LIN {X 0,Y 362.1,Z 510.041,A -85,B 0,C 180,E1 -13379.691,E2 -13379.691} C_VEL
LIN {X 0,Y 361.308,Z 518.217,A -85,B 0,C 180,E1 -13381.227,E2 -13381.227} C_VEL
LIN {X 0,Y 359.207,Z 536.983,A -85,B 0,C 180,E1 -13384.658,E2 -13384.658} C_VEL
LIN {X 0,Y 359.602,Z 541.842,A -85,B 0,C 180,E1 -13385.074,E2 -13385.074} C_VEL
LIN {X 0,Y 360.933,Z 553.52,A -85,B 0,C 180,E1 -13385.902,E2 -13385.902} C_VEL
LIN {X 0,Y 363.229,Z 569.599,A -85,B 0,C 180,E1 -13386.676,E2 -13386.676} C_VEL
LIN {X 0,Y 364.954,Z 589.975,A -85,B 0,C 180,E1 -13387.487,E2 -13387.487} C_VEL
LIN {X 0,Y 365.399,Z 602.018,A -85,B 0,C 180,E1 -13387.902,E2 -13387.902} C_VEL
LIN {X 0,Y 363.82,Z 641.826,A -85,B 0,C 180,E1 -13388.948,E2 -13388.948} C_VEL
LIN {X 0,Y 363.382,Z 660.329,A -85,B 0,C 180,E1 -13389.366,E2 -13389.366} C_VEL
LIN {X 0,Y 362.094,Z 683.326,A -85,B 0,C 180,E1 -13390.216,E2 -13390.216} C_VEL
LIN {X 0,Y 360.889,Z 696.981,A -85,B 0,C 180,E1 -13390.96,E2 -13390.96} C_VEL
LIN {X 0,Y 359.746,Z 709.851,A -85,B 0,C 180,E1 -13391.931,E2 -13391.931} C_VEL
LIN {X 0,Y 358.479,Z 721.302,A -85,B 0,C 180,E1 -13393.043,E2 -13393.043} C_VEL
LIN {X 0,Y 357.211,Z 731.941,A -85,B 0,C 180,E1 -13394.329,E2 -13394.329} C_VEL
LIN {X 0,Y 356.095,Z 741.238,A -85,B 0,C 180,E1 -13395.716,E2 -13395.716} C_VEL
LIN {X 0,Y 355.187,Z 750.5,A -85,B 0,C 180,E1 -13397.427,E2 -13397.427} C_VEL
LIN {X 0,Y 354.364,Z 757.955,A -85,B 0,C 180,E1 -13399.138,E2 -13399.138} C_VEL
LIN {X 0,Y 353.848,Z 763.907,A -85,B 0,C 180,E1 -13400.855,E2 -13400.855} C_VEL
LIN {X 0,Y 353.526,Z 768.592,A -85,B 0,C 180,E1 -13402.574,E2 -13402.574} C_VEL
LIN {X 0,Y 353.412,Z 772.146,A -85,B 0,C 180,E1 -13404.292,E2 -13404.292} C_VEL
LIN {X 0,Y 353.428,Z 773.933,A -85,B 0,C 180,E1 -13405.436,E2 -13405.436} C_VEL
LIN {X 0,Y 353.398,Z 775.272,A -85,B 0,C 180,E1 -13406.578,E2 -13406.578} C_VEL
LIN {X 0,Y 353.5,Z 776.131,A -85,B 0,C 180,E1 -13407.719,E2 -13407.719} C_VEL
LIN {X 0,Y 353.555,Z 776.567,A -85,B 0,C 180,E1 -13408.859,E2 -13408.859} C_VEL
LIN {X 0,Y 353.604,Z 776.578,A -85,B 0,C 180,E1 -13409.998,E2 -13409.998} C_VEL
LIN {X 0,Y 353.57,Z 776.1,A -85,B 0,C 180,E1 -13411.137,E2 -13411.137} C_VEL
LIN {X 0,Y 353.576,Z 775.182,A -85,B 0,C 180,E1 -13412.276,E2 -13412.276} C_VEL
LIN {X 0,Y 353.45,Z 773.823,A -85,B 0,C 180,E1 -13413.418,E2 -13413.418} C_VEL
LIN {X 0,Y 353.526,Z 770.885,A -85,B 0,C 180,E1 -13415.131,E2 -13415.131} C_VEL
LIN {X 0,Y 353.504,Z 766.785,A -85,B 0,C 180,E1 -13416.849,E2 -13416.849} C_VEL
LIN {X 0,Y 353.73,Z 760.366,A -85,B 0,C 180,E1 -13418.856,E2 -13418.856} C_VEL
LIN {X 0,Y 354.077,Z 753.304,A -85,B 0,C 180,E1 -13420.578,E2 -13420.578} C_VEL
LIN {X 0,Y 354.591,Z 746.042,A -85,B 0,C 180,E1 -13422.01,E2 -13422.01} C_VEL
LIN {X 0,Y 355.295,Z 737.187,A -85,B 0,C 180,E1 -13423.438,E2 -13423.438} C_VEL
LIN {X 0,Y 355.944,Z 727.505,A -85,B 0,C 180,E1 -13424.717,E2 -13424.717} C_VEL
LIN {X 0,Y 356.758,Z 716.84,A -85,B 0,C 180,E1 -13425.861,E2 -13425.861} C_VEL
LIN {X 0,Y 357.66,Z 705.092,A -85,B 0,C 180,E1 -13426.846,E2 -13426.846} C_VEL
LIN {X 0,Y 359.257,Z 682.161,A -85,B 0,C 180,E1 -13428.312,E2 -13428.312} C_VEL
LIN {X 0,Y 360.052,Z 669.426,A -85,B 0,C 180,E1 -13428.934,E2 -13428.934} C_VEL
LIN {X 0,Y 360.522,Z 656.027,A -85,B 0,C 180,E1 -13429.351,E2 -13429.351} C_VEL
LIN {X 0,Y 361.316,Z 597.635,A -85,B 0,C 180,E1 -13430.517,E2 -13430.517} C_VEL
LIN {X 0,Y 357.035,Z 553.883,A -85,B 0,C 180,E1 -13431.65,E2 -13431.65} C_VEL
LIN {X 0,Y 356.733,Z 547.954,A -85,B 0,C 180,E1 -13431.944,E2 -13431.944} C_VEL
LIN {X 0,Y 358.479,Z 525.594,A -85,B 0,C 180,E1 -13435.86,E2 -13435.86} C_VEL
LIN {X 0,Y 360.164,Z 506.756,A -85,B 0,C 180,E1 -13439.196,E2 -13439.196} C_VEL
LIN {X 0,Y 359.872,Z 503.178,A -85,B 0,C 180,E1 -13439.865,E2 -13439.865} C_VEL
LIN {X 0,Y 356.669,Z 488.438,A -85,B 0,C 180,E1 -13442.808,E2 -13442.808} C_VEL
LIN {X 0,Y 354.865,Z 480.388,A -85,B 0,C 180,E1 -13444.535,E2 -13444.535} C_VEL
LIN {X 0,Y 354.786,Z 480.291,A -85,B 0,C 180,E1 -13447.882,E2 -13447.882} C_VEL
LIN {X 0,Y 354.763,Z 480.29,A -85,B 0,C 180,E1 -13451.166,E2 -13451.166} C_VEL
LIN {X 0,Y 354.754,Z 480.295,A -85,B 0,C 180,E1 -13454.504,E2 -13454.504} C_VEL
LIN {X 0,Y 354.781,Z 480.289,A -85,B 0,C 180,E1 -13457.66,E2 -13457.66} C_VEL
LIN {X 0,Y 354.775,Z 480.291,A -85,B 0,C 180,E1 -13460.66,E2 -13460.66} C_VEL
LIN {X 0,Y 354.811,Z 480.291,A -85,B 0,C 180,E1 -13464.299,E2 -13464.299} C_VEL
LIN {X 0,Y 354.776,Z 480.29,A -85,B 0,C 180,E1 -13467.665,E2 -13467.665} C_VEL
LIN {X 0,Y 354.818,Z 480.287,A -85,B 0,C 180,E1 -13470.631,E2 -13470.631} C_VEL
LIN {X 0,Y 354.887,Z 480.279,A -85,B 0,C 180,E1 -13474.171,E2 -13474.171} C_VEL
LIN {X 0,Y 354.822,Z 480.285,A -85,B 0,C 180,E1 -13477.893,E2 -13477.893} C_VEL
LIN {X 0,Y 354.91,Z 480.274,A -85,B 0,C 180,E1 -13481.891,E2 -13481.891} C_VEL
LIN {X 0,Y 354.93,Z 480.272,A -85,B 0,C 180,E1 -13485.98,E2 -13485.98} C_VEL
LIN {X 0,Y 354.965,Z 480.266,A -85,B 0,C 180,E1 -13489.735,E2 -13489.735} C_VEL
LIN {X 0,Y 355.1,Z 480.25,A -85,B 0,C 180,E1 -13492.036,E2 -13492.036} C_VEL
LIN {X 0,Y 355.076,Z 480.256,A -85,B 0,C 180,E1 -13494.32,E2 -13494.32} C_VEL
LIN {X 0,Y 355.23,Z 480.232,A -85,B 0,C 180,E1 -13497.732,E2 -13497.732} C_VEL
LIN {X 0,Y 355.383,Z 480.214,A -85,B 0,C 180,E1 -13500,E2 -13500} C_VEL
LIN {X 0,Y 355.231,Z 480.235,A -85,B 0,C 180,E1 -13502.267,E2 -13502.267} C_VEL
LIN {X 0,Y 355.122,Z 480.25,A -85,B 0,C 180,E1 -13506.819,E2 -13506.819} C_VEL
LIN {X 0,Y 355.001,Z 480.262,A -85,B 0,C 180,E1 -13509.112,E2 -13509.112} C_VEL
LIN {X 0,Y 354.907,Z 480.278,A -85,B 0,C 180,E1 -13512.581,E2 -13512.581} C_VEL
LIN {X 0,Y 354.876,Z 480.278,A -85,B 0,C 180,E1 -13516.096,E2 -13516.096} C_VEL
LIN {X 0,Y 354.892,Z 480.278,A -85,B 0,C 180,E1 -13518.472,E2 -13518.472} C_VEL
LIN {X 0,Y 354.821,Z 480.284,A -85,B 0,C 180,E1 -13522.106,E2 -13522.106} C_VEL
LIN {X 0,Y 354.886,Z 480.275,A -85,B 0,C 180,E1 -13525.828,E2 -13525.828} C_VEL
LIN {X 0,Y 354.84,Z 480.281,A -85,B 0,C 180,E1 -13529.679,E2 -13529.679} C_VEL
LIN {X 0,Y 354.793,Z 480.287,A -85,B 0,C 180,E1 -13533.703,E2 -13533.703} C_VEL
LIN {X 0,Y 354.786,Z 480.29,A -85,B 0,C 180,E1 -13536.46,E2 -13536.46} C_VEL
LIN {X 0,Y 354.812,Z 480.285,A -85,B 0,C 180,E1 -13539.425,E2 -13539.425} C_VEL
LIN {X 0,Y 354.779,Z 480.295,A -85,B 0,C 180,E1 -13542.869,E2 -13542.869} C_VEL
LIN {X 0,Y 354.841,Z 480.281,A -85,B 0,C 180,E1 -13546.118,E2 -13546.118} C_VEL
LIN {X 0,Y 354.846,Z 480.284,A -85,B 0,C 180,E1 -13549.19,E2 -13549.19} C_VEL
LIN {X 0,Y 354.806,Z 480.286,A -85,B 0,C 180,E1 -13552.402,E2 -13552.402} C_VEL
LIN {X 0,Y 354.803,Z 480.292,A -85,B 0,C 180,E1 -13554.943,E2 -13554.943} C_VEL
LIN {X 0,Y 354.784,Z 480.289,A -85,B 0,C 180,E1 -13558.407,E2 -13558.407} C_VEL
LIN {X 0,Y 354.841,Z 480.281,A -85,B 0,C 180,E1 -13561.621,E2 -13561.621} C_VEL
LIN {X 0,Y 354.892,Z 480.274,A -85,B 0,C 180,E1 -13564.174,E2 -13564.174} C_VEL
LIN {X 0,Y 354.828,Z 480.282,A -85,B 0,C 180,E1 -13567.896,E2 -13567.896} C_VEL
LIN {X 0,Y 354.917,Z 480.271,A -85,B 0,C 180,E1 -13571.893,E2 -13571.893} C_VEL
LIN {X 0,Y 354.938,Z 480.269,A -85,B 0,C 180,E1 -13575.983,E2 -13575.983} C_VEL
LIN {X 0,Y 354.974,Z 480.269,A -85,B 0,C 180,E1 -13579.738,E2 -13579.738} C_VEL
LIN {X 0,Y 355.126,Z 480.377,A -85,B 0,C 180,E1 -13582.826,E2 -13582.826} C_VEL
LIN {X 0,Y 355.316,Z 481.259,A -85,B 0,C 180,E1 -13583.026,E2 -13583.026} C_VEL
LIN {X 0,Y 362.099,Z 500.146,A -85,B 0,C 180,E1 -13583.792,E2 -13583.792} C_VEL
LIN {X 0,Y 361.485,Z 558.412,A -85,B 0,C 180,E1 -13584.965,E2 -13584.965} C_VEL
LIN {X 0,Y 361.353,Z 571.995,A -85,B 0,C 180,E1 -13585.396,E2 -13585.396} C_VEL
LIN {X 0,Y 361.076,Z 584.594,A -85,B 0,C 180,E1 -13586.026,E2 -13586.026} C_VEL
LIN {X 0,Y 360.556,Z 597.464,A -85,B 0,C 180,E1 -13586.929,E2 -13586.929} C_VEL
LIN {X 0,Y 359.941,Z 608.176,A -85,B 0,C 180,E1 -13587.904,E2 -13587.904} C_VEL
LIN {X 0,Y 359.185,Z 618.721,A -85,B 0,C 180,E1 -13589.104,E2 -13589.104} C_VEL
LIN {X 0,Y 358.367,Z 628.913,A -85,B 0,C 180,E1 -13590.563,E2 -13590.563} C_VEL
LIN {X 0,Y 357.609,Z 636.954,A -85,B 0,C 180,E1 -13591.973,E2 -13591.973} C_VEL
LIN {X 0,Y 356.893,Z 644.84,A -85,B 0,C 180,E1 -13593.671,E2 -13593.671} C_VEL
LIN {X 0,Y 356.349,Z 650.193,A -85,B 0,C 180,E1 -13595.094,E2 -13595.094} C_VEL
LIN {X 0,Y 355.867,Z 655.436,A -85,B 0,C 180,E1 -13596.807,E2 -13596.807} C_VEL
LIN {X 0,Y 355.462,Z 659.828,A -85,B 0,C 180,E1 -13598.673,E2 -13598.673} C_VEL
LIN {X 0,Y 355.184,Z 662.585,A -85,B 0,C 180,E1 -13600.26,E2 -13600.26} C_VEL
LIN {X 0,Y 355.045,Z 664.08,A -85,B 0,C 180,E1 -13601.419,E2 -13601.419} C_VEL
LIN {X 0,Y 355.044,Z 665.804,A -85,B 0,C 180,E1 -13603.743,E2 -13603.743} C_VEL
LIN {X 0,Y 355.098,Z 666.085,A -85,B 0,C 180,E1 -13604.911,E2 -13604.911} C_VEL
LIN {X 0,Y 355.215,Z 665.916,A -85,B 0,C 180,E1 -13606.083,E2 -13606.083} C_VEL
LIN {X 0,Y 355.368,Z 665.349,A -85,B 0,C 180,E1 -13607.258,E2 -13607.258} C_VEL
LIN {X 0,Y 355.643,Z 664.352,A -85,B 0,C 180,E1 -13608.461,E2 -13608.461} C_VEL
LIN {X 0,Y 355.959,Z 662.949,A -85,B 0,C 180,E1 -13609.614,E2 -13609.614} C_VEL
LIN {X 0,Y 356.56,Z 659.952,A -85,B 0,C 180,E1 -13611.388,E2 -13611.388} C_VEL
LIN {X 0,Y 357.35,Z 655.819,A -85,B 0,C 180,E1 -13613.164,E2 -13613.164} C_VEL
LIN {X 0,Y 358.298,Z 650.412,A -85,B 0,C 180,E1 -13614.945,E2 -13614.945} C_VEL
LIN {X 0,Y 359.447,Z 643.529,A -85,B 0,C 180,E1 -13616.726,E2 -13616.726} C_VEL
LIN {X 0,Y 360.613,Z 635.638,A -85,B 0,C 180,E1 -13618.357,E2 -13618.357} C_VEL
LIN {X 0,Y 361.847,Z 626.608,A -85,B 0,C 180,E1 -13619.85,E2 -13619.85} C_VEL
LIN {X 0,Y 362.979,Z 616.583,A -85,B 0,C 180,E1 -13621.196,E2 -13621.196} C_VEL
LIN {X 0,Y 364.189,Z 605.349,A -85,B 0,C 180,E1 -13622.384,E2 -13622.384} C_VEL
LIN {X 0,Y 364.443,Z 601.847,A -85,B 0,C 180,E1 -13622.703,E2 -13622.703} C_VEL
LIN {X 0,Y 364.337,Z 599.564,A -85,B 0,C 180,E1 -13622.919,E2 -13622.919} C_VEL
LIN {X 0,Y 362.891,Z 595.342,A -85,B 0,C 180,E1 -13623.393,E2 -13623.393} C_VEL
LIN {X 0,Y 359.587,Z 588.061,A -85,B 0,C 180,E1 -13624.197,E2 -13624.197} C_VEL
LIN {X 0,Y 359.103,Z 584.474,A -85,B 0,C 180,E1 -13624.462,E2 -13624.462} C_VEL
LIN {X 0,Y 359.463,Z 571.812,A -85,B 0,C 180,E1 -13625.075,E2 -13625.075} C_VEL
LIN {X 0,Y 359.573,Z 558.207,A -85,B 0,C 180,E1 -13625.48,E2 -13625.48} C_VEL
LIN {X 0,Y 360.319,Z 507.281,A -85,B 0,C 180,E1 -13626.549,E2 -13626.549} C_VEL
LIN {X 0,Y 352.428,Z 490.788,A -85,B 0,C 180,E1 -13627.596,E2 -13627.596} C_VEL
LIN {X 0,Y 348.024,Z 482.285,A -85,B 0,C 180,E1 -13628.212,E2 -13628.212} C_VEL
LIN {X 0,Y 347.78,Z 481.299,A -85,B 0,C 180,E1 -13628.444,E2 -13628.444} C_VEL
LIN {X 0,Y 347.755,Z 481.16,A -85,B 0,C 180,E1 -13631.832,E2 -13631.832} C_VEL
LIN {X 0,Y 347.71,Z 481.173,A -85,B 0,C 180,E1 -13635.028,E2 -13635.028} C_VEL
LIN {X 0,Y 347.82,Z 481.408,A -85,B 0,C 180,E1 -13636.936,E2 -13636.936} C_VEL
LIN {X 0,Y 351.431,Z 497.302,A -85,B 0,C 180,E1 -13640.213,E2 -13640.213} C_VEL
LIN {X 0,Y 352.832,Z 505.673,A -85,B 0,C 180,E1 -13641.868,E2 -13641.868} C_VEL
LIN {X 0,Y 351.854,Z 524.218,A -85,B 0,C 180,E1 -13645.237,E2 -13645.237} C_VEL
LIN {X 0,Y 355.268,Z 547.014,A -85,B 0,C 180,E1 -13646.026,E2 -13646.026} C_VEL
LIN {X 0,Y 352.98,Z 635.486,A -85,B 0,C 180,E1 -13648.239,E2 -13648.239} C_VEL
LIN {X 0,Y 352.469,Z 648.238,A -85,B 0,C 180,E1 -13648.774,E2 -13648.774} C_VEL
LIN {X 0,Y 351.763,Z 662.108,A -85,B 0,C 180,E1 -13649.619,E2 -13649.619} C_VEL
LIN {X 0,Y 351.002,Z 674.363,A -85,B 0,C 180,E1 -13650.623,E2 -13650.623} C_VEL
LIN {X 0,Y 350.092,Z 686.153,A -85,B 0,C 180,E1 -13651.857,E2 -13651.857} C_VEL
LIN {X 0,Y 349.229,Z 696.648,A -85,B 0,C 180,E1 -13653.239,E2 -13653.239} C_VEL
LIN {X 0,Y 348.378,Z 707.013,A -85,B 0,C 180,E1 -13654.936,E2 -13654.936} C_VEL
LIN {X 0,Y 347.758,Z 714.569,A -85,B 0,C 180,E1 -13656.476,E2 -13656.476} C_VEL
LIN {X 0,Y 347.18,Z 721.867,A -85,B 0,C 180,E1 -13658.32,E2 -13658.32} C_VEL
LIN {X 0,Y 346.818,Z 726.724,A -85,B 0,C 180,E1 -13659.85,E2 -13659.85} C_VEL
LIN {X 0,Y 346.503,Z 731.293,A -85,B 0,C 180,E1 -13661.677,E2 -13661.677} C_VEL
LIN {X 0,Y 346.306,Z 734.624,A -85,B 0,C 180,E1 -13663.494,E2 -13663.494} C_VEL
LIN {X 0,Y 346.177,Z 736.196,A -85,B 0,C 180,E1 -13664.697,E2 -13664.697} C_VEL
LIN {X 0,Y 346.252,Z 737.936,A -85,B 0,C 180,E1 -13666.982,E2 -13666.982} C_VEL
LIN {X 0,Y 346.292,Z 738.175,A -85,B 0,C 180,E1 -13668.291,E2 -13668.291} C_VEL
LIN {X 0,Y 346.341,Z 737.941,A -85,B 0,C 180,E1 -13669.477,E2 -13669.477} C_VEL
LIN {X 0,Y 346.511,Z 737.282,A -85,B 0,C 180,E1 -13670.662,E2 -13670.662} C_VEL
LIN {X 0,Y 346.735,Z 736.138,A -85,B 0,C 180,E1 -13671.844,E2 -13671.844} C_VEL
LIN {X 0,Y 347.109,Z 733.621,A -85,B 0,C 180,E1 -13673.607,E2 -13673.607} C_VEL
LIN {X 0,Y 347.593,Z 730.052,A -85,B 0,C 180,E1 -13675.361,E2 -13675.361} C_VEL
LIN {X 0,Y 348.301,Z 725.327,A -85,B 0,C 180,E1 -13677.109,E2 -13677.109} C_VEL
LIN {X 0,Y 349.188,Z 719.362,A -85,B 0,C 180,E1 -13678.847,E2 -13678.847} C_VEL
LIN {X 0,Y 350.351,Z 711.877,A -85,B 0,C 180,E1 -13680.575,E2 -13680.575} C_VEL
LIN {X 0,Y 351.69,Z 702.532,A -85,B 0,C 180,E1 -13682.291,E2 -13682.291} C_VEL
LIN {X 0,Y 352.98,Z 692.894,A -85,B 0,C 180,E1 -13683.711,E2 -13683.711} C_VEL
LIN {X 0,Y 354.3,Z 682.127,A -85,B 0,C 180,E1 -13684.979,E2 -13684.979} C_VEL
LIN {X 0,Y 355.51,Z 670.303,A -85,B 0,C 180,E1 -13686.1,E2 -13686.1} C_VEL
LIN {X 0,Y 356.608,Z 657.741,A -85,B 0,C 180,E1 -13687.005,E2 -13687.005} C_VEL
LIN {X 0,Y 357.436,Z 644.738,A -85,B 0,C 180,E1 -13687.698,E2 -13687.698} C_VEL
LIN {X 0,Y 358.056,Z 630.868,A -85,B 0,C 180,E1 -13688.182,E2 -13688.182} C_VEL
LIN {X 0,Y 361.68,Z 550.068,A -85,B 0,C 180,E1 -13690.392,E2 -13690.392} C_VEL
LIN {X 0,Y 358.98,Z 536.542,A -85,B 0,C 180,E1 -13691.139,E2 -13691.139} C_VEL
LIN {X 0,Y 356.986,Z 528.228,A -85,B 0,C 180,E1 -13691.678,E2 -13691.678} C_VEL
LIN {X 0,Y 357.932,Z 515.694,A -85,B 0,C 180,E1 -13694.026,E2 -13694.026} C_VEL
LIN {X 0,Y 356.287,Z 506.932,A -85,B 0,C 180,E1 -13696.032,E2 -13696.032} C_VEL
LIN {X 0,Y 354.005,Z 498.233,A -85,B 0,C 180,E1 -13698.19,E2 -13698.19} C_VEL
LIN {X 0,Y 351.666,Z 491.215,A -85,B 0,C 180,E1 -13700.064,E2 -13700.064} C_VEL
LIN {X 0,Y 348.904,Z 484.236,A -85,B 0,C 180,E1 -13702.088,E2 -13702.088} C_VEL
LIN {X 0,Y 347.802,Z 481.291,A -85,B 0,C 180,E1 -13703.088,E2 -13703.088} C_VEL
LIN {X 0,Y 347.839,Z 481.156,A -85,B 0,C 180,E1 -13706.392,E2 -13706.392} C_VEL
LIN {X 0,Y 347.759,Z 481.165,A -85,B 0,C 180,E1 -13710.347,E2 -13710.347} C_VEL
LIN {X 0,Y 347.757,Z 481.164,A -85,B 0,C 180,E1 -13714.043,E2 -13714.043} C_VEL
LIN {X 0,Y 347.77,Z 481.166,A -85,B 0,C 180,E1 -13717.32,E2 -13717.32} C_VEL
LIN {X 0,Y 347.741,Z 481.166,A -85,B 0,C 180,E1 -13720.296,E2 -13720.296} C_VEL
LIN {X 0,Y 347.732,Z 481.171,A -85,B 0,C 180,E1 -13723.407,E2 -13723.407} C_VEL
LIN {X 0,Y 347.734,Z 481.168,A -85,B 0,C 180,E1 -13726.685,E2 -13726.685} C_VEL
LIN {X 0,Y 347.756,Z 481.155,A -85,B 0,C 180,E1 -13730.172,E2 -13730.172} C_VEL
LIN {X 0,Y 347.826,Z 481.368,A -85,B 0,C 180,E1 -13732.301,E2 -13732.301} C_VEL
LIN {X 0,Y 350.98,Z 492.829,A -85,B 0,C 180,E1 -13735.184,E2 -13735.184} C_VEL
LIN {X 0,Y 354.051,Z 505.655,A -85,B 0,C 180,E1 -13738.155,E2 -13738.155} C_VEL
LIN {X 0,Y 355.2,Z 511.151,A -85,B 0,C 180,E1 -13739.368,E2 -13739.368} C_VEL
LIN {X 0,Y 355.151,Z 514.431,A -85,B 0,C 180,E1 -13740.02,E2 -13740.02} C_VEL
LIN {X 0,Y 352.808,Z 534.057,A -85,B 0,C 180,E1 -13743.691,E2 -13743.691} C_VEL
LIN {X 0,Y 354.361,Z 550.862,A -85,B 0,C 180,E1 -13745.073,E2 -13745.073} C_VEL
LIN {X 0,Y 356.839,Z 567.558,A -85,B 0,C 180,E1 -13745.946,E2 -13745.946} C_VEL
LIN {X 0,Y 358.367,Z 583.9,A -85,B 0,C 180,E1 -13746.658,E2 -13746.658} C_VEL
LIN {X 0,Y 359.28,Z 601.18,A -85,B 0,C 180,E1 -13747.316,E2 -13747.316} C_VEL
LIN {X 0,Y 357.163,Z 651.513,A -85,B 0,C 180,E1 -13748.688,E2 -13748.688} C_VEL
LIN {X 0,Y 356.174,Z 675.049,A -85,B 0,C 180,E1 -13749.383,E2 -13749.383} C_VEL
LIN {X 0,Y 355.277,Z 688.078,A -85,B 0,C 180,E1 -13749.971,E2 -13749.971} C_VEL
LIN {X 0,Y 354.094,Z 700.242,A -85,B 0,C 180,E1 -13750.731,E2 -13750.731} C_VEL
LIN {X 0,Y 352.899,Z 712.253,A -85,B 0,C 180,E1 -13751.718,E2 -13751.718} C_VEL
LIN {X 0,Y 351.576,Z 723.182,A -85,B 0,C 180,E1 -13752.85,E2 -13752.85} C_VEL
LIN {X 0,Y 350.259,Z 733.453,A -85,B 0,C 180,E1 -13754.177,E2 -13754.177} C_VEL
LIN {X 0,Y 349.042,Z 743.13,A -85,B 0,C 180,E1 -13755.718,E2 -13755.718} C_VEL
LIN {X 0,Y 348.064,Z 751.871,A -85,B 0,C 180,E1 -13757.462,E2 -13757.462} C_VEL
LIN {X 0,Y 347.27,Z 758.972,A -85,B 0,C 180,E1 -13759.209,E2 -13759.209} C_VEL
LIN {X 0,Y 346.672,Z 765.481,A -85,B 0,C 180,E1 -13761.253,E2 -13761.253} C_VEL
LIN {X 0,Y 346.416,Z 769.706,A -85,B 0,C 180,E1 -13763.006,E2 -13763.006} C_VEL
LIN {X 0,Y 346.32,Z 771.894,A -85,B 0,C 180,E1 -13764.174,E2 -13764.174} C_VEL
LIN {X 0,Y 346.335,Z 773.649,A -85,B 0,C 180,E1 -13765.342,E2 -13765.342} C_VEL
LIN {X 0,Y 346.313,Z 774.928,A -85,B 0,C 180,E1 -13766.508,E2 -13766.508} C_VEL
LIN {X 0,Y 346.399,Z 775.759,A -85,B 0,C 180,E1 -13767.673,E2 -13767.673} C_VEL
LIN {X 0,Y 346.487,Z 776.17,A -85,B 0,C 180,E1 -13768.836,E2 -13768.836} C_VEL
LIN {X 0,Y 346.533,Z 776.135,A -85,B 0,C 180,E1 -13769.998,E2 -13769.998} C_VEL
LIN {X 0,Y 346.504,Z 775.611,A -85,B 0,C 180,E1 -13771.16,E2 -13771.16} C_VEL
LIN {X 0,Y 346.492,Z 774.661,A -85,B 0,C 180,E1 -13772.323,E2 -13772.323} C_VEL
LIN {X 0,Y 346.364,Z 773.257,A -85,B 0,C 180,E1 -13773.488,E2 -13773.488} C_VEL
LIN {X 0,Y 346.434,Z 770.239,A -85,B 0,C 180,E1 -13775.236,E2 -13775.236} C_VEL
LIN {X 0,Y 346.416,Z 766.039,A -85,B 0,C 180,E1 -13776.99,E2 -13776.99} C_VEL
LIN {X 0,Y 346.674,Z 759.52,A -85,B 0,C 180,E1 -13779.037,E2 -13779.037} C_VEL
LIN {X 0,Y 347.028,Z 752.324,A -85,B 0,C 180,E1 -13780.795,E2 -13780.795} C_VEL
LIN {X 0,Y 347.691,Z 743.241,A -85,B 0,C 180,E1 -13782.548,E2 -13782.548} C_VEL
LIN {X 0,Y 348.554,Z 733.916,A -85,B 0,C 180,E1 -13784,E2 -13784} C_VEL
LIN {X 0,Y 349.104,Z 724.751,A -85,B 0,C 180,E1 -13785.169,E2 -13785.169} C_VEL
LIN {X 0,Y 350.034,Z 713.509,A -85,B 0,C 180,E1 -13786.323,E2 -13786.323} C_VEL
LIN {X 0,Y 350.86,Z 700.933,A -85,B 0,C 180,E1 -13787.333,E2 -13787.333} C_VEL
LIN {X 0,Y 352.677,Z 677.371,A -85,B 0,C 180,E1 -13788.817,E2 -13788.817} C_VEL
LIN {X 0,Y 353.418,Z 663.783,A -85,B 0,C 180,E1 -13789.416,E2 -13789.416} C_VEL
LIN {X 0,Y 353.806,Z 649.393,A -85,B 0,C 180,E1 -13789.785,E2 -13789.785} C_VEL
LIN {X 0,Y 354.472,Z 597.967,A -85,B 0,C 180,E1 -13790.827,E2 -13790.827} C_VEL
LIN {X 0,Y 350.181,Z 553.243,A -85,B 0,C 180,E1 -13792.002,E2 -13792.002} C_VEL
LIN {X 0,Y 349.796,Z 546.99,A -85,B 0,C 180,E1 -13792.323,E2 -13792.323} C_VEL
LIN {X 0,Y 351.533,Z 525.872,A -85,B 0,C 180,E1 -13796.091,E2 -13796.091} C_VEL
LIN {X 0,Y 353.168,Z 508.484,A -85,B 0,C 180,E1 -13799.239,E2 -13799.239} C_VEL
LIN {X 0,Y 353.06,Z 505.286,A -85,B 0,C 180,E1 -13799.842,E2 -13799.842} C_VEL
LIN {X 0,Y 349.9,Z 490.522,A -85,B 0,C 180,E1 -13802.839,E2 -13802.839} C_VEL
LIN {X 0,Y 347.827,Z 481.272,A -85,B 0,C 180,E1 -13804.848,E2 -13804.848} C_VEL
LIN {X 0,Y 347.723,Z 481.169,A -85,B 0,C 180,E1 -13808.794,E2 -13808.794} C_VEL
LIN {X 0,Y 347.736,Z 481.169,A -85,B 0,C 180,E1 -13811.829,E2 -13811.829} C_VEL
LIN {X 0,Y 347.696,Z 481.171,A -85,B 0,C 180,E1 -13815.025,E2 -13815.025} C_VEL
LIN {X 0,Y 347.737,Z 481.17,A -85,B 0,C 180,E1 -13818.396,E2 -13818.396} C_VEL
LIN {X 0,Y 347.753,Z 481.167,A -85,B 0,C 180,E1 -13822.012,E2 -13822.012} C_VEL
LIN {X 0,Y 347.734,Z 481.166,A -85,B 0,C 180,E1 -13825.534,E2 -13825.534} C_VEL
LIN {X 0,Y 347.75,Z 481.165,A -85,B 0,C 180,E1 -13829.652,E2 -13829.652} C_VEL
LIN {X 0,Y 347.819,Z 481.155,A -85,B 0,C 180,E1 -13833.606,E2 -13833.606} C_VEL
LIN {X 0,Y 347.776,Z 481.165,A -85,B 0,C 180,E1 -13836.161,E2 -13836.161} C_VEL
LIN {X 0,Y 347.8,Z 481.159,A -85,B 0,C 180,E1 -13839.908,E2 -13839.908} C_VEL
LIN {X 0,Y 347.853,Z 481.156,A -85,B 0,C 180,E1 -13842.358,E2 -13842.358} C_VEL
LIN {X 0,Y 347.884,Z 481.149,A -85,B 0,C 180,E1 -13845.97,E2 -13845.97} C_VEL
LIN {X 0,Y 347.916,Z 481.142,A -85,B 0,C 180,E1 -13849.525,E2 -13849.525} C_VEL
LIN {X 0,Y 348.06,Z 481.126,A -85,B 0,C 180,E1 -13851.874,E2 -13851.874} C_VEL
LIN {X 0,Y 348.051,Z 481.13,A -85,B 0,C 180,E1 -13854.205,E2 -13854.205} C_VEL
LIN {X 0,Y 348.192,Z 481.108,A -85,B 0,C 180,E1 -13857.686,E2 -13857.686} C_VEL
LIN {X 0,Y 348.332,Z 481.092,A -85,B 0,C 180,E1 -13860,E2 -13860} C_VEL
LIN {X 0,Y 348.193,Z 481.112,A -85,B 0,C 180,E1 -13862.313,E2 -13862.313} C_VEL
LIN {X 0,Y 348.091,Z 481.123,A -85,B 0,C 180,E1 -13866.958,E2 -13866.958} C_VEL
LIN {X 0,Y 347.953,Z 481.138,A -85,B 0,C 180,E1 -13869.298,E2 -13869.298} C_VEL
LIN {X 0,Y 347.876,Z 481.153,A -85,B 0,C 180,E1 -13872.84,E2 -13872.84} C_VEL
LIN {X 0,Y 347.825,Z 481.158,A -85,B 0,C 180,E1 -13876.432,E2 -13876.432} C_VEL
LIN {X 0,Y 347.842,Z 481.156,A -85,B 0,C 180,E1 -13878.861,E2 -13878.861} C_VEL
LIN {X 0,Y 347.76,Z 481.167,A -85,B 0,C 180,E1 -13882.58,E2 -13882.58} C_VEL
LIN {X 0,Y 347.799,Z 481.16,A -85,B 0,C 180,E1 -13885.109,E2 -13885.109} C_VEL
LIN {X 0,Y 347.797,Z 481.157,A -85,B 0,C 180,E1 -13887.695,E2 -13887.695} C_VEL
LIN {X 0,Y 347.75,Z 481.165,A -85,B 0,C 180,E1 -13890.347,E2 -13890.347} C_VEL
LIN {X 0,Y 347.732,Z 481.169,A -85,B 0,C 180,E1 -13894.465,E2 -13894.465} C_VEL
LIN {X 0,Y 347.762,Z 481.162,A -85,B 0,C 180,E1 -13897.99,E2 -13897.99} C_VEL
LIN {X 0,Y 347.739,Z 481.165,A -85,B 0,C 180,E1 -13901.831,E2 -13901.831} C_VEL
LIN {X 0,Y 347.786,Z 481.164,A -85,B 0,C 180,E1 -13905.013,E2 -13905.013} C_VEL
LIN {X 0,Y 347.774,Z 481.163,A -85,B 0,C 180,E1 -13908.392,E2 -13908.392} C_VEL
LIN {X 0,Y 347.772,Z 481.16,A -85,B 0,C 180,E1 -13912.011,E2 -13912.011} C_VEL
LIN {X 0,Y 347.735,Z 481.167,A -85,B 0,C 180,E1 -13915.538,E2 -13915.538} C_VEL
LIN {X 0,Y 347.755,Z 481.164,A -85,B 0,C 180,E1 -13919.655,E2 -13919.655} C_VEL
LIN {X 0,Y 347.843,Z 481.155,A -85,B 0,C 180,E1 -13922.747,E2 -13922.747} C_VEL
LIN {X 0,Y 347.781,Z 481.16,A -85,B 0,C 180,E1 -13926.164,E2 -13926.164} C_VEL
LIN {X 0,Y 347.806,Z 481.157,A -85,B 0,C 180,E1 -13929.911,E2 -13929.911} C_VEL
LIN {X 0,Y 347.861,Z 481.151,A -85,B 0,C 180,E1 -13932.361,E2 -13932.361} C_VEL
LIN {X 0,Y 347.893,Z 481.146,A -85,B 0,C 180,E1 -13935.973,E2 -13935.973} C_VEL
LIN {X 0,Y 347.925,Z 481.147,A -85,B 0,C 180,E1 -13939.528,E2 -13939.528} C_VEL
LIN {X 0,Y 348.101,Z 481.261,A -85,B 0,C 180,E1 -13942.461,E2 -13942.461} C_VEL
LIN {X 0,Y 348.275,Z 482.132,A -85,B 0,C 180,E1 -13942.66,E2 -13942.66} C_VEL
LIN {X 0,Y 354.817,Z 500.197,A -85,B 0,C 180,E1 -13943.422,E2 -13943.422} C_VEL
LIN {X 0,Y 355.393,Z 501.827,A -85,B 0,C 180,E1 -13943.486,E2 -13943.486} C_VEL
LIN {X 0,Y 354.671,Z 557.634,A -85,B 0,C 180,E1 -13944.621,E2 -13944.621} C_VEL
LIN {X 0,Y 354.607,Z 570.905,A -85,B 0,C 180,E1 -13945.022,E2 -13945.022} C_VEL
LIN {X 0,Y 354.344,Z 584.159,A -85,B 0,C 180,E1 -13945.665,E2 -13945.665} C_VEL
LIN {X 0,Y 353.856,Z 595.708,A -85,B 0,C 180,E1 -13946.444,E2 -13946.444} C_VEL
LIN {X 0,Y 353.234,Z 606.942,A -85,B 0,C 180,E1 -13947.436,E2 -13947.436} C_VEL
LIN {X 0,Y 352.392,Z 618.377,A -85,B 0,C 180,E1 -13948.716,E2 -13948.716} C_VEL
LIN {X 0,Y 351.654,Z 627.602,A -85,B 0,C 180,E1 -13950.002,E2 -13950.002} C_VEL
LIN {X 0,Y 350.859,Z 636.042,A -85,B 0,C 180,E1 -13951.437,E2 -13951.437} C_VEL
LIN {X 0,Y 350.065,Z 644.254,A -85,B 0,C 180,E1 -13953.167,E2 -13953.167} C_VEL
LIN {X 0,Y 349.375,Z 650.895,A -85,B 0,C 180,E1 -13954.906,E2 -13954.906} C_VEL
LIN {X 0,Y 348.809,Z 656.97,A -85,B 0,C 180,E1 -13956.945,E2 -13956.945} C_VEL
LIN {X 0,Y 348.409,Z 660.991,A -85,B 0,C 180,E1 -13958.734,E2 -13958.734} C_VEL
LIN {X 0,Y 348.137,Z 663.875,A -85,B 0,C 180,E1 -13960.47,E2 -13960.47} C_VEL
LIN {X 0,Y 347.952,Z 666.283,A -85,B 0,C 180,E1 -13962.839,E2 -13962.839} C_VEL
LIN {X 0,Y 348.018,Z 666.942,A -85,B 0,C 180,E1 -13964.229,E2 -13964.229} C_VEL
LIN {X 0,Y 348.233,Z 666.831,A -85,B 0,C 180,E1 -13966.414,E2 -13966.414} C_VEL
LIN {X 0,Y 348.685,Z 665.293,A -85,B 0,C 180,E1 -13968.682,E2 -13968.682} C_VEL
LIN {X 0,Y 349.085,Z 663.628,A -85,B 0,C 180,E1 -13970.016,E2 -13970.016} C_VEL
LIN {X 0,Y 349.765,Z 660.503,A -85,B 0,C 180,E1 -13971.824,E2 -13971.824} C_VEL
LIN {X 0,Y 350.596,Z 656.236,A -85,B 0,C 180,E1 -13973.637,E2 -13973.637} C_VEL
LIN {X 0,Y 351.632,Z 650.697,A -85,B 0,C 180,E1 -13975.446,E2 -13975.446} C_VEL
LIN {X 0,Y 352.843,Z 643.603,A -85,B 0,C 180,E1 -13977.268,E2 -13977.268} C_VEL
LIN {X 0,Y 354.22,Z 634.768,A -85,B 0,C 180,E1 -13979.047,E2 -13979.047} C_VEL
LIN {X 0,Y 355.554,Z 625.147,A -85,B 0,C 180,E1 -13980.598,E2 -13980.598} C_VEL
LIN {X 0,Y 356.642,Z 615.779,A -85,B 0,C 180,E1 -13981.814,E2 -13981.814} C_VEL
LIN {X 0,Y 357.875,Z 604.013,A -85,B 0,C 180,E1 -13983.023,E2 -13983.023} C_VEL
LIN {X 0,Y 358.68,Z 592.578,A -85,B 0,C 180,E1 -13983.949,E2 -13983.949} C_VEL
LIN {X 0,Y 359.103,Z 584.474,A -85,B 0,C 180,E1 -13984.462,E2 -13984.462} C_VEL
LIN {X 0,Y 358.639,Z 580.826,A -85,B 0,C 180,E1 -13984.715,E2 -13984.715} C_VEL
LIN {X 0,Y 353.839,Z 569.554,A -85,B 0,C 180,E1 -13985.63,E2 -13985.63} C_VEL
LIN {X 0,Y 353.24,Z 565.762,A -85,B 0,C 180,E1 -13985.8,E2 -13985.8} C_VEL
LIN {X 0,Y 353.596,Z 531.568,A -85,B 0,C 180,E1 -13986.565,E2 -13986.565} C_VEL
LIN {X 0,Y 354.086,Z 509.377,A -85,B 0,C 180,E1 -13987.027,E2 -13987.027} C_VEL
LIN {X 0,Y 345.254,Z 491.331,A -85,B 0,C 180,E1 -13988.235,E2 -13988.235} C_VEL
LIN {X 0,Y 340.891,Z 482.935,A -85,B 0,C 180,E1 -13988.887,E2 -13988.887} C_VEL
LIN {X 0,Y 340.72,Z 482.127,A -85,B 0,C 180,E1 -13989.127,E2 -13989.127} C_VEL
LIN {X 0,Y 340.68,Z 482.039,A -85,B 0,C 180,E1 -13992.906,E2 -13992.906} C_VEL
LIN {X 0,Y 340.73,Z 482.222,A -85,B 0,C 180,E1 -13996.574,E2 -13996.574} C_VEL
LIN {X 0,Y 344.424,Z 498.211,A -85,B 0,C 180,E1 -13999.926,E2 -13999.926} C_VEL
LIN {X 0,Y 345.944,Z 507.075,A -85,B 0,C 180,E1 -14001.712,E2 -14001.712} C_VEL
LIN {X 0,Y 344.985,Z 524.509,A -85,B 0,C 180,E1 -14004.902,E2 -14004.902} C_VEL
LIN {X 0,Y 348.438,Z 548.358,A -85,B 0,C 180,E1 -14005.738,E2 -14005.738} C_VEL
LIN {X 0,Y 346.083,Z 635.054,A -85,B 0,C 180,E1 -14007.959,E2 -14007.959} C_VEL
LIN {X 0,Y 345.569,Z 648.231,A -85,B 0,C 180,E1 -14008.513,E2 -14008.513} C_VEL
LIN {X 0,Y 344.825,Z 662.067,A -85,B 0,C 180,E1 -14009.368,E2 -14009.368} C_VEL
LIN {X 0,Y 344.113,Z 673.594,A -85,B 0,C 180,E1 -14010.313,E2 -14010.313} C_VEL
LIN {X 0,Y 343.256,Z 684.703,A -85,B 0,C 180,E1 -14011.47,E2 -14011.47} C_VEL
LIN {X 0,Y 342.35,Z 695.204,A -85,B 0,C 180,E1 -14012.822,E2 -14012.822} C_VEL
LIN {X 0,Y 341.533,Z 705.036,A -85,B 0,C 180,E1 -14014.397,E2 -14014.397} C_VEL
LIN {X 0,Y 340.855,Z 713.039,A -85,B 0,C 180,E1 -14015.97,E2 -14015.97} C_VEL
LIN {X 0,Y 340.231,Z 720.78,A -85,B 0,C 180,E1 -14017.854,E2 -14017.854} C_VEL
LIN {X 0,Y 339.833,Z 725.931,A -85,B 0,C 180,E1 -14019.417,E2 -14019.417} C_VEL
LIN {X 0,Y 339.476,Z 730.774,A -85,B 0,C 180,E1 -14021.284,E2 -14021.284} C_VEL
LIN {X 0,Y 339.245,Z 734.365,A -85,B 0,C 180,E1 -14023.141,E2 -14023.141} C_VEL
LIN {X 0,Y 339.105,Z 736.138,A -85,B 0,C 180,E1 -14024.37,E2 -14024.37} C_VEL
LIN {X 0,Y 339.092,Z 737.416,A -85,B 0,C 180,E1 -14025.599,E2 -14025.599} C_VEL
LIN {X 0,Y 339.163,Z 738.252,A -85,B 0,C 180,E1 -14026.891,E2 -14026.891} C_VEL
LIN {X 0,Y 339.191,Z 738.602,A -85,B 0,C 180,E1 -14028.042,E2 -14028.042} C_VEL
LIN {X 0,Y 339.239,Z 738.507,A -85,B 0,C 180,E1 -14029.255,E2 -14029.255} C_VEL
LIN {X 0,Y 339.419,Z 737.964,A -85,B 0,C 180,E1 -14030.466,E2 -14030.466} C_VEL
LIN {X 0,Y 339.643,Z 737.006,A -85,B 0,C 180,E1 -14031.672,E2 -14031.672} C_VEL
LIN {X 0,Y 339.929,Z 735.479,A -85,B 0,C 180,E1 -14032.941,E2 -14032.941} C_VEL
LIN {X 0,Y 340.374,Z 732.613,A -85,B 0,C 180,E1 -14034.669,E2 -14034.669} C_VEL
LIN {X 0,Y 340.948,Z 728.574,A -85,B 0,C 180,E1 -14036.455,E2 -14036.455} C_VEL
LIN {X 0,Y 341.994,Z 722.326,A -85,B 0,C 180,E1 -14038.528,E2 -14038.528} C_VEL
LIN {X 0,Y 343.111,Z 715.44,A -85,B 0,C 180,E1 -14040.294,E2 -14040.294} C_VEL
LIN {X 0,Y 344.515,Z 706.683,A -85,B 0,C 180,E1 -14042.076,E2 -14042.076} C_VEL
LIN {X 0,Y 345.937,Z 697.123,A -85,B 0,C 180,E1 -14043.64,E2 -14043.64} C_VEL
LIN {X 0,Y 347.41,Z 686.133,A -85,B 0,C 180,E1 -14045.078,E2 -14045.078} C_VEL
LIN {X 0,Y 348.687,Z 675.163,A -85,B 0,C 180,E1 -14046.22,E2 -14046.22} C_VEL
LIN {X 0,Y 349.898,Z 662.933,A -85,B 0,C 180,E1 -14047.212,E2 -14047.212} C_VEL
LIN {X 0,Y 350.92,Z 650.198,A -85,B 0,C 180,E1 -14047.987,E2 -14047.987} C_VEL
LIN {X 0,Y 351.562,Z 638.031,A -85,B 0,C 180,E1 -14048.515,E2 -14048.515} C_VEL
LIN {X 0,Y 355.668,Z 550.588,A -85,B 0,C 180,E1 -14051.018,E2 -14051.018} C_VEL
LIN {X 0,Y 352.239,Z 534.43,A -85,B 0,C 180,E1 -14051.991,E2 -14051.991} C_VEL
LIN {X 0,Y 350.863,Z 528.524,A -85,B 0,C 180,E1 -14052.432,E2 -14052.432} C_VEL
LIN {X 0,Y 351.685,Z 518.286,A -85,B 0,C 180,E1 -14054.389,E2 -14054.389} C_VEL
LIN {X 0,Y 349.892,Z 508.809,A -85,B 0,C 180,E1 -14056.621,E2 -14056.621} C_VEL
LIN {X 0,Y 347.535,Z 500.116,A -85,B 0,C 180,E1 -14058.879,E2 -14058.879} C_VEL
LIN {X 0,Y 345.132,Z 493.085,A -85,B 0,C 180,E1 -14060.876,E2 -14060.876} C_VEL
LIN {X 0,Y 342.031,Z 485.308,A -85,B 0,C 180,E1 -14063.3,E2 -14063.3} C_VEL
LIN {X 0,Y 340.807,Z 482.226,A -85,B 0,C 180,E1 -14064.403,E2 -14064.403} C_VEL
LIN {X 0,Y 340.786,Z 482.037,A -85,B 0,C 180,E1 -14067.525,E2 -14067.525} C_VEL
LIN {X 0,Y 340.707,Z 482.048,A -85,B 0,C 180,E1 -14071.044,E2 -14071.044} C_VEL
LIN {X 0,Y 340.727,Z 482.043,A -85,B 0,C 180,E1 -14075.278,E2 -14075.278} C_VEL
LIN {X 0,Y 340.718,Z 482.041,A -85,B 0,C 180,E1 -14078.385,E2 -14078.385} C_VEL
LIN {X 0,Y 340.708,Z 482.042,A -85,B 0,C 180,E1 -14082.045,E2 -14082.045} C_VEL
LIN {X 0,Y 340.66,Z 482.048,A -85,B 0,C 180,E1 -14086.226,E2 -14086.226} C_VEL
LIN {X 0,Y 340.697,Z 482.043,A -85,B 0,C 180,E1 -14089.752,E2 -14089.752} C_VEL
LIN {X 0,Y 340.747,Z 482.224,A -85,B 0,C 180,E1 -14091.664,E2 -14091.664} C_VEL
LIN {X 0,Y 343.656,Z 492.596,A -85,B 0,C 180,E1 -14094.382,E2 -14094.382} C_VEL
LIN {X 0,Y 346.874,Z 505.664,A -85,B 0,C 180,E1 -14097.525,E2 -14097.525} C_VEL
LIN {X 0,Y 348.512,Z 513.941,A -85,B 0,C 180,E1 -14099.389,E2 -14099.389} C_VEL
LIN {X 0,Y 346.716,Z 528.522,A -85,B 0,C 180,E1 -14102.209,E2 -14102.209} C_VEL
LIN {X 0,Y 346.473,Z 531.431,A -85,B 0,C 180,E1 -14102.679,E2 -14102.679} C_VEL
LIN {X 0,Y 348.226,Z 549.933,A -85,B 0,C 180,E1 -14104.282,E2 -14104.282} C_VEL
LIN {X 0,Y 350.157,Z 562.98,A -85,B 0,C 180,E1 -14105.048,E2 -14105.048} C_VEL
LIN {X 0,Y 352.021,Z 579.57,A -85,B 0,C 180,E1 -14105.843,E2 -14105.843} C_VEL
LIN {X 0,Y 353.231,Z 601.413,A -85,B 0,C 180,E1 -14106.722,E2 -14106.722} C_VEL
LIN {X 0,Y 349.922,Z 673.807,A -85,B 0,C 180,E1 -14108.805,E2 -14108.805} C_VEL
LIN {X 0,Y 348.932,Z 687.676,A -85,B 0,C 180,E1 -14109.436,E2 -14109.436} C_VEL
LIN {X 0,Y 347.694,Z 699.766,A -85,B 0,C 180,E1 -14110.208,E2 -14110.208} C_VEL
LIN {X 0,Y 346.397,Z 711.678,A -85,B 0,C 180,E1 -14111.209,E2 -14111.209} C_VEL
LIN {X 0,Y 345.019,Z 722.554,A -85,B 0,C 180,E1 -14112.36,E2 -14112.36} C_VEL
LIN {X 0,Y 343.485,Z 733.553,A -85,B 0,C 180,E1 -14113.811,E2 -14113.811} C_VEL
LIN {X 0,Y 342.153,Z 743.498,A -85,B 0,C 180,E1 -14115.448,E2 -14115.448} C_VEL
LIN {X 0,Y 341.13,Z 751.984,A -85,B 0,C 180,E1 -14117.203,E2 -14117.203} C_VEL
LIN {X 0,Y 340.267,Z 758.962,A -85,B 0,C 180,E1 -14118.984,E2 -14118.984} C_VEL
LIN {X 0,Y 339.612,Z 765.331,A -85,B 0,C 180,E1 -14121.069,E2 -14121.069} C_VEL
LIN {X 0,Y 339.344,Z 769.494,A -85,B 0,C 180,E1 -14122.86,E2 -14122.86} C_VEL
LIN {X 0,Y 339.241,Z 771.657,A -85,B 0,C 180,E1 -14124.052,E2 -14124.052} C_VEL
LIN {X 0,Y 339.245,Z 773.373,A -85,B 0,C 180,E1 -14125.245,E2 -14125.245} C_VEL
LIN {X 0,Y 339.231,Z 774.593,A -85,B 0,C 180,E1 -14126.435,E2 -14126.435} C_VEL
LIN {X 0,Y 339.299,Z 775.39,A -85,B 0,C 180,E1 -14127.624,E2 -14127.624} C_VEL
LIN {X 0,Y 339.42,Z 775.771,A -85,B 0,C 180,E1 -14128.812,E2 -14128.812} C_VEL
LIN {X 0,Y 339.464,Z 775.67,A -85,B 0,C 180,E1 -14129.998,E2 -14129.998} C_VEL
LIN {X 0,Y 339.439,Z 775.115,A -85,B 0,C 180,E1 -14131.184,E2 -14131.184} C_VEL
LIN {X 0,Y 339.395,Z 774.132,A -85,B 0,C 180,E1 -14132.372,E2 -14132.372} C_VEL
LIN {X 0,Y 339.283,Z 772.666,A -85,B 0,C 180,E1 -14133.561,E2 -14133.561} C_VEL
LIN {X 0,Y 339.344,Z 769.573,A -85,B 0,C 180,E1 -14135.346,E2 -14135.346} C_VEL
LIN {X 0,Y 339.344,Z 765.287,A -85,B 0,C 180,E1 -14137.136,E2 -14137.136} C_VEL
LIN {X 0,Y 339.566,Z 759.716,A -85,B 0,C 180,E1 -14138.928,E2 -14138.928} C_VEL
LIN {X 0,Y 339.908,Z 752.669,A -85,B 0,C 180,E1 -14140.722,E2 -14140.722} C_VEL
LIN {X 0,Y 340.466,Z 745.434,A -85,B 0,C 180,E1 -14142.213,E2 -14142.213} C_VEL
LIN {X 0,Y 341.221,Z 736.613,A -85,B 0,C 180,E1 -14143.699,E2 -14143.699} C_VEL
LIN {X 0,Y 341.852,Z 727.388,A -85,B 0,C 180,E1 -14144.978,E2 -14144.978} C_VEL
LIN {X 0,Y 342.737,Z 716.33,A -85,B 0,C 180,E1 -14146.221,E2 -14146.221} C_VEL
LIN {X 0,Y 343.706,Z 704.69,A -85,B 0,C 180,E1 -14147.245,E2 -14147.245} C_VEL
LIN {X 0,Y 345.153,Z 685.745,A -85,B 0,C 180,E1 -14148.549,E2 -14148.549} C_VEL
LIN {X 0,Y 346.049,Z 672.94,A -85,B 0,C 180,E1 -14149.307,E2 -14149.307} C_VEL
LIN {X 0,Y 346.721,Z 659.327,A -85,B 0,C 180,E1 -14149.845,E2 -14149.845} C_VEL
LIN {X 0,Y 347.294,Z 627.077,A -85,B 0,C 180,E1 -14150.55,E2 -14150.55} C_VEL
LIN {X 0,Y 347.577,Z 597.817,A -85,B 0,C 180,E1 -14151.159,E2 -14151.159} C_VEL
LIN {X 0,Y 343.241,Z 552.073,A -85,B 0,C 180,E1 -14152.389,E2 -14152.389} C_VEL
LIN {X 0,Y 342.873,Z 545.857,A -85,B 0,C 180,E1 -14152.722,E2 -14152.722} C_VEL
LIN {X 0,Y 344.726,Z 524.458,A -85,B 0,C 180,E1 -14156.646,E2 -14156.646} C_VEL
LIN {X 0,Y 346.24,Z 509.1,A -85,B 0,C 180,E1 -14159.485,E2 -14159.485} C_VEL
LIN {X 0,Y 345.895,Z 505.522,A -85,B 0,C 180,E1 -14160.188,E2 -14160.188} C_VEL
LIN {X 0,Y 342.587,Z 490.09,A -85,B 0,C 180,E1 -14163.407,E2 -14163.407} C_VEL
LIN {X 0,Y 340.779,Z 482.144,A -85,B 0,C 180,E1 -14165.188,E2 -14165.188} C_VEL
LIN {X 0,Y 340.686,Z 482.048,A -85,B 0,C 180,E1 -14168.38,E2 -14168.38} C_VEL
LIN {X 0,Y 340.685,Z 482.049,A -85,B 0,C 180,E1 -14172.042,E2 -14172.042} C_VEL
LIN {X 0,Y 340.643,Z 482.055,A -85,B 0,C 180,E1 -14176.225,E2 -14176.225} C_VEL
LIN {X 0,Y 340.664,Z 482.049,A -85,B 0,C 180,E1 -14179.754,E2 -14179.754} C_VEL
LIN {X 0,Y 340.692,Z 482.043,A -85,B 0,C 180,E1 -14183.256,E2 -14183.256} C_VEL
LIN {X 0,Y 340.682,Z 482.048,A -85,B 0,C 180,E1 -14186.152,E2 -14186.152} C_VEL
LIN {X 0,Y 340.773,Z 482.038,A -85,B 0,C 180,E1 -14190.332,E2 -14190.332} C_VEL
LIN {X 0,Y 340.791,Z 482.031,A -85,B 0,C 180,E1 -14193.018,E2 -14193.018} C_VEL
LIN {X 0,Y 340.716,Z 482.042,A -85,B 0,C 180,E1 -14196.926,E2 -14196.926} C_VEL
LIN {X 0,Y 340.778,Z 482.035,A -85,B 0,C 180,E1 -14200.732,E2 -14200.732} C_VEL
LIN {X 0,Y 340.773,Z 482.033,A -85,B 0,C 180,E1 -14203.218,E2 -14203.218} C_VEL
LIN {X 0,Y 340.831,Z 482.027,A -85,B 0,C 180,E1 -14206.89,E2 -14206.89} C_VEL
LIN {X 0,Y 340.915,Z 482.02,A -85,B 0,C 180,E1 -14210.507,E2 -14210.507} C_VEL
LIN {X 0,Y 341.061,Z 482,A -85,B 0,C 180,E1 -14212.897,E2 -14212.897} C_VEL
LIN {X 0,Y 341.154,Z 481.984,A -85,B 0,C 180,E1 -14217.638,E2 -14217.638} C_VEL
LIN {X 0,Y 341.282,Z 481.969,A -85,B 0,C 180,E1 -14220,E2 -14220} C_VEL
LIN {X 0,Y 341.155,Z 481.989,A -85,B 0,C 180,E1 -14222.361,E2 -14222.361} C_VEL
LIN {X 0,Y 341.06,Z 481.997,A -85,B 0,C 180,E1 -14227.102,E2 -14227.102} C_VEL
LIN {X 0,Y 340.857,Z 482.028,A -85,B 0,C 180,E1 -14230.694,E2 -14230.694} C_VEL
LIN {X 0,Y 340.849,Z 482.027,A -85,B 0,C 180,E1 -14234.325,E2 -14234.325} C_VEL
LIN {X 0,Y 340.824,Z 482.03,A -85,B 0,C 180,E1 -14238.467,E2 -14238.467} C_VEL
LIN {X 0,Y 340.74,Z 482.037,A -85,B 0,C 180,E1 -14241.857,E2 -14241.857} C_VEL
LIN {X 0,Y 340.759,Z 482.035,A -85,B 0,C 180,E1 -14245.665,E2 -14245.665} C_VEL
LIN {X 0,Y 340.728,Z 482.039,A -85,B 0,C 180,E1 -14248.32,E2 -14248.32} C_VEL
LIN {X 0,Y 340.69,Z 482.047,A -85,B 0,C 180,E1 -14251.045,E2 -14251.045} C_VEL
LIN {X 0,Y 340.705,Z 482.043,A -85,B 0,C 180,E1 -14255.28,E2 -14255.28} C_VEL
LIN {X 0,Y 340.698,Z 482.043,A -85,B 0,C 180,E1 -14258.387,E2 -14258.387} C_VEL
LIN {X 0,Y 340.688,Z 482.044,A -85,B 0,C 180,E1 -14262.047,E2 -14262.047} C_VEL
LIN {X 0,Y 340.71,Z 482.042,A -85,B 0,C 180,E1 -14265.469,E2 -14265.469} C_VEL
LIN {X 0,Y 340.715,Z 482.045,A -85,B 0,C 180,E1 -14268.698,E2 -14268.698} C_VEL
LIN {X 0,Y 340.736,Z 482.036,A -85,B 0,C 180,E1 -14271.776,E2 -14271.776} C_VEL
LIN {X 0,Y 340.714,Z 482.04,A -85,B 0,C 180,E1 -14275.597,E2 -14275.597} C_VEL
LIN {X 0,Y 340.695,Z 482.049,A -85,B 0,C 180,E1 -14278.958,E2 -14278.958} C_VEL
LIN {X 0,Y 340.769,Z 482.032,A -85,B 0,C 180,E1 -14282.476,E2 -14282.476} C_VEL
LIN {X 0,Y 340.749,Z 482.038,A -85,B 0,C 180,E1 -14285.64,E2 -14285.64} C_VEL
LIN {X 0,Y 340.739,Z 482.04,A -85,B 0,C 180,E1 -14289.476,E2 -14289.476} C_VEL
LIN {X 0,Y 340.852,Z 482.024,A -85,B 0,C 180,E1 -14291.986,E2 -14291.986} C_VEL
LIN {X 0,Y 340.864,Z 482.022,A -85,B 0,C 180,E1 -14295.707,E2 -14295.707} C_VEL
LIN {X 0,Y 340.867,Z 482.026,A -85,B 0,C 180,E1 -14299.308,E2 -14299.308} C_VEL
LIN {X 0,Y 341.07,Z 482.207,A -85,B 0,C 180,E1 -14302.122,E2 -14302.122} C_VEL
LIN {X 0,Y 341.325,Z 483.305,A -85,B 0,C 180,E1 -14302.313,E2 -14302.313} C_VEL
LIN {X 0,Y 347.525,Z 500.147,A -85,B 0,C 180,E1 -14303.033,E2 -14303.033} C_VEL
LIN {X 0,Y 348.652,Z 503.424,A -85,B 0,C 180,E1 -14303.164,E2 -14303.164} C_VEL
LIN {X 0,Y 347.857,Z 557.282,A -85,B 0,C 180,E1 -14304.277,E2 -14304.277} C_VEL
LIN {X 0,Y 347.831,Z 570.897,A -85,B 0,C 180,E1 -14304.676,E2 -14304.676} C_VEL
LIN {X 0,Y 347.564,Z 583.701,A -85,B 0,C 180,E1 -14305.29,E2 -14305.29} C_VEL
LIN {X 0,Y 347.067,Z 595.605,A -85,B 0,C 180,E1 -14306.083,E2 -14306.083} C_VEL
LIN {X 0,Y 346.435,Z 607.115,A -85,B 0,C 180,E1 -14307.095,E2 -14307.095} C_VEL
LIN {X 0,Y 345.578,Z 618.683,A -85,B 0,C 180,E1 -14308.4,E2 -14308.4} C_VEL
LIN {X 0,Y 344.729,Z 628.763,A -85,B 0,C 180,E1 -14309.822,E2 -14309.822} C_VEL
LIN {X 0,Y 343.799,Z 638.072,A -85,B 0,C 180,E1 -14311.466,E2 -14311.466} C_VEL
LIN {X 0,Y 343.009,Z 646.105,A -85,B 0,C 180,E1 -14313.232,E2 -14313.232} C_VEL
LIN {X 0,Y 342.423,Z 651.583,A -85,B 0,C 180,E1 -14314.711,E2 -14314.711} C_VEL
LIN {X 0,Y 341.89,Z 656.942,A -85,B 0,C 180,E1 -14316.494,E2 -14316.494} C_VEL
LIN {X 0,Y 341.462,Z 661.145,A -85,B 0,C 180,E1 -14318.286,E2 -14318.286} C_VEL
LIN {X 0,Y 341.222,Z 663.383,A -85,B 0,C 180,E1 -14319.486,E2 -14319.486} C_VEL
LIN {X 0,Y 341.076,Z 665.128,A -85,B 0,C 180,E1 -14320.689,E2 -14320.689} C_VEL
LIN {X 0,Y 340.936,Z 667.423,A -85,B 0,C 180,E1 -14323.108,E2 -14323.108} C_VEL
LIN {X 0,Y 341,Z 667.944,A -85,B 0,C 180,E1 -14324.382,E2 -14324.382} C_VEL
LIN {X 0,Y 341.252,Z 667.749,A -85,B 0,C 180,E1 -14326.76,E2 -14326.76} C_VEL
LIN {X 0,Y 341.752,Z 666.217,A -85,B 0,C 180,E1 -14328.921,E2 -14328.921} C_VEL
LIN {X 0,Y 342.441,Z 663.347,A -85,B 0,C 180,E1 -14331.05,E2 -14331.05} C_VEL
LIN {X 0,Y 343.215,Z 659.721,A -85,B 0,C 180,E1 -14332.898,E2 -14332.898} C_VEL
LIN {X 0,Y 344.222,Z 654.886,A -85,B 0,C 180,E1 -14334.745,E2 -14334.745} C_VEL
LIN {X 0,Y 345.375,Z 648.679,A -85,B 0,C 180,E1 -14336.597,E2 -14336.597} C_VEL
LIN {X 0,Y 346.586,Z 642.229,A -85,B 0,C 180,E1 -14338.131,E2 -14338.131} C_VEL
LIN {X 0,Y 347.798,Z 634.41,A -85,B 0,C 180,E1 -14339.669,E2 -14339.669} C_VEL
LIN {X 0,Y 349.151,Z 624.586,A -85,B 0,C 180,E1 -14341.221,E2 -14341.221} C_VEL
LIN {X 0,Y 350.335,Z 615.007,A -85,B 0,C 180,E1 -14342.441,E2 -14342.441} C_VEL
LIN {X 0,Y 351.478,Z 604.339,A -85,B 0,C 180,E1 -14343.532,E2 -14343.532} C_VEL
LIN {X 0,Y 352.357,Z 591.911,A -85,B 0,C 180,E1 -14344.527,E2 -14344.527} C_VEL
LIN {X 0,Y 352.98,Z 578.947,A -85,B 0,C 180,E1 -14345.282,E2 -14345.282} C_VEL
LIN {X 0,Y 353.193,Z 567.1,A -85,B 0,C 180,E1 -14345.761,E2 -14345.761} C_VEL
LIN {X 0,Y 353.24,Z 565.762,A -85,B 0,C 180,E1 -14345.8,E2 -14345.8} C_VEL
LIN {X 0,Y 352.618,Z 561.928,A -85,B 0,C 180,E1 -14345.955,E2 -14345.955} C_VEL
LIN {X 0,Y 347.567,Z 550.153,A -85,B 0,C 180,E1 -14346.654,E2 -14346.654} C_VEL
LIN {X 0,Y 347.04,Z 546.301,A -85,B 0,C 180,E1 -14346.788,E2 -14346.788} C_VEL
LIN {X 0,Y 347.739,Z 511.353,A -85,B 0,C 180,E1 -14347.538,E2 -14347.538} C_VEL
LIN {X 0,Y 338.618,Z 492.795,A -85,B 0,C 180,E1 -14348.835,E2 -14348.835} C_VEL
LIN {X 0,Y 333.872,Z 483.991,A -85,B 0,C 180,E1 -14349.553,E2 -14349.553} C_VEL
LIN {X 0,Y 333.68,Z 483.008,A -85,B 0,C 180,E1 -14349.804,E2 -14349.804} C_VEL
LIN {X 0,Y 333.637,Z 482.915,A -85,B 0,C 180,E1 -14352.501,E2 -14352.501} C_VEL
LIN {X 0,Y 333.658,Z 483.082,A -85,B 0,C 180,E1 -14356.23,E2 -14356.23} C_VEL
LIN {X 0,Y 337.298,Z 498.738,A -85,B 0,C 180,E1 -14359.56,E2 -14359.56} C_VEL
LIN {X 0,Y 339.04,Z 508.533,A -85,B 0,C 180,E1 -14361.547,E2 -14361.547} C_VEL
LIN {X 0,Y 338.135,Z 524.817,A -85,B 0,C 180,E1 -14364.555,E2 -14364.555} C_VEL
LIN {X 0,Y 341.618,Z 548.559,A -85,B 0,C 180,E1 -14365.411,E2 -14365.411} C_VEL
LIN {X 0,Y 339.144,Z 636.353,A -85,B 0,C 180,E1 -14367.749,E2 -14367.749} C_VEL
LIN {X 0,Y 338.544,Z 649.592,A -85,B 0,C 180,E1 -14368.339,E2 -14368.339} C_VEL
LIN {X 0,Y 337.819,Z 662.815,A -85,B 0,C 180,E1 -14369.183,E2 -14369.183} C_VEL
LIN {X 0,Y 337.112,Z 674.257,A -85,B 0,C 180,E1 -14370.15,E2 -14370.15} C_VEL
LIN {X 0,Y 336.146,Z 686.079,A -85,B 0,C 180,E1 -14371.419,E2 -14371.419} C_VEL
LIN {X 0,Y 335.218,Z 696.866,A -85,B 0,C 180,E1 -14372.871,E2 -14372.871} C_VEL
LIN {X 0,Y 334.323,Z 707.14,A -85,B 0,C 180,E1 -14374.601,E2 -14374.601} C_VEL
LIN {X 0,Y 333.725,Z 714.322,A -85,B 0,C 180,E1 -14376.085,E2 -14376.085} C_VEL
LIN {X 0,Y 333.184,Z 720.74,A -85,B 0,C 180,E1 -14377.686,E2 -14377.686} C_VEL
LIN {X 0,Y 332.702,Z 726.88,A -85,B 0,C 180,E1 -14379.602,E2 -14379.602} C_VEL
LIN {X 0,Y 332.349,Z 731.612,A -85,B 0,C 180,E1 -14381.507,E2 -14381.507} C_VEL
LIN {X 0,Y 332.2,Z 734.092,A -85,B 0,C 180,E1 -14382.772,E2 -14382.772} C_VEL
LIN {X 0,Y 332.036,Z 736.001,A -85,B 0,C 180,E1 -14384.029,E2 -14384.029} C_VEL
LIN {X 0,Y 332.013,Z 737.454,A -85,B 0,C 180,E1 -14385.285,E2 -14385.285} C_VEL
LIN {X 0,Y 332.092,Z 738.56,A -85,B 0,C 180,E1 -14386.784,E2 -14386.784} C_VEL
LIN {X 0,Y 332.14,Z 739.019,A -85,B 0,C 180,E1 -14389.022,E2 -14389.022} C_VEL
LIN {X 0,Y 332.298,Z 738.653,A -85,B 0,C 180,E1 -14390.259,E2 -14390.259} C_VEL
LIN {X 0,Y 332.528,Z 737.815,A -85,B 0,C 180,E1 -14391.493,E2 -14391.493} C_VEL
LIN {X 0,Y 332.864,Z 736.336,A -85,B 0,C 180,E1 -14392.918,E2 -14392.918} C_VEL
LIN {X 0,Y 333.467,Z 732.692,A -85,B 0,C 180,E1 -14395.165,E2 -14395.165} C_VEL
LIN {X 0,Y 334.158,Z 728.522,A -85,B 0,C 180,E1 -14396.986,E2 -14396.986} C_VEL
LIN {X 0,Y 335.126,Z 723.121,A -85,B 0,C 180,E1 -14398.799,E2 -14398.799} C_VEL
LIN {X 0,Y 336.309,Z 716.387,A -85,B 0,C 180,E1 -14400.599,E2 -14400.599} C_VEL
LIN {X 0,Y 337.774,Z 707.937,A -85,B 0,C 180,E1 -14402.385,E2 -14402.385} C_VEL
LIN {X 0,Y 339.133,Z 699.33,A -85,B 0,C 180,E1 -14403.862,E2 -14403.862} C_VEL
LIN {X 0,Y 340.673,Z 688.726,A -85,B 0,C 180,E1 -14405.327,E2 -14405.327} C_VEL
LIN {X 0,Y 342.225,Z 676.772,A -85,B 0,C 180,E1 -14406.634,E2 -14406.634} C_VEL
LIN {X 0,Y 343.485,Z 664.974,A -85,B 0,C 180,E1 -14407.643,E2 -14407.643} C_VEL
LIN {X 0,Y 344.665,Z 651.684,A -85,B 0,C 180,E1 -14408.502,E2 -14408.502} C_VEL
LIN {X 0,Y 345.366,Z 639.221,A -85,B 0,C 180,E1 -14409.074,E2 -14409.074} C_VEL
LIN {X 0,Y 349.859,Z 552.178,A -85,B 0,C 180,E1 -14411.629,E2 -14411.629} C_VEL
LIN {X 0,Y 346.271,Z 535.247,A -85,B 0,C 180,E1 -14412.707,E2 -14412.707} C_VEL
LIN {X 0,Y 344.811,Z 529.088,A -85,B 0,C 180,E1 -14413.181,E2 -14413.181} C_VEL
LIN {X 0,Y 345.519,Z 521.156,A -85,B 0,C 180,E1 -14414.73,E2 -14414.73} C_VEL
LIN {X 0,Y 343.893,Z 512.085,A -85,B 0,C 180,E1 -14416.932,E2 -14416.932} C_VEL
LIN {X 0,Y 341.613,Z 503.549,A -85,B 0,C 180,E1 -14419.219,E2 -14419.219} C_VEL
LIN {X 0,Y 338.917,Z 495.666,A -85,B 0,C 180,E1 -14421.589,E2 -14421.589} C_VEL
LIN {X 0,Y 335.481,Z 487.092,A -85,B 0,C 180,E1 -14424.441,E2 -14424.441} C_VEL
LIN {X 0,Y 333.77,Z 483.117,A -85,B 0,C 180,E1 -14426.004,E2 -14426.004} C_VEL
LIN {X 0,Y 333.699,Z 482.918,A -85,B 0,C 180,E1 -14428.974,E2 -14428.974} C_VEL
LIN {X 0,Y 333.653,Z 482.923,A -85,B 0,C 180,E1 -14432.586,E2 -14432.586} C_VEL
LIN {X 0,Y 333.685,Z 482.917,A -85,B 0,C 180,E1 -14436.138,E2 -14436.138} C_VEL
LIN {X 0,Y 333.655,Z 482.925,A -85,B 0,C 180,E1 -14439.192,E2 -14439.192} C_VEL
LIN {X 0,Y 333.641,Z 482.922,A -85,B 0,C 180,E1 -14442.499,E2 -14442.499} C_VEL
LIN {X 0,Y 333.605,Z 482.928,A -85,B 0,C 180,E1 -14445.954,E2 -14445.954} C_VEL
LIN {X 0,Y 333.656,Z 482.926,A -85,B 0,C 180,E1 -14449.314,E2 -14449.314} C_VEL
LIN {X 0,Y 333.715,Z 483.082,A -85,B 0,C 180,E1 -14450.998,E2 -14450.998} C_VEL
LIN {X 0,Y 336.8,Z 493.976,A -85,B 0,C 180,E1 -14453.96,E2 -14453.96} C_VEL
LIN {X 0,Y 339.951,Z 506.815,A -85,B 0,C 180,E1 -14457.132,E2 -14457.132} C_VEL
LIN {X 0,Y 341.663,Z 515.069,A -85,B 0,C 180,E1 -14459.051,E2 -14459.051} C_VEL
LIN {X 0,Y 341.224,Z 519.942,A -85,B 0,C 180,E1 -14460.036,E2 -14460.036} C_VEL
LIN {X 0,Y 340.314,Z 527.095,A -85,B 0,C 180,E1 -14461.387,E2 -14461.387} C_VEL
LIN {X 0,Y 341.666,Z 542.977,A -85,B 0,C 180,E1 -14462.926,E2 -14462.926} C_VEL
LIN {X 0,Y 342.511,Z 552.071,A -85,B 0,C 180,E1 -14463.684,E2 -14463.684} C_VEL
LIN {X 0,Y 344.982,Z 569.029,A -85,B 0,C 180,E1 -14464.647,E2 -14464.647} C_VEL
LIN {X 0,Y 346.465,Z 585.95,A -85,B 0,C 180,E1 -14465.452,E2 -14465.452} C_VEL
LIN {X 0,Y 347.168,Z 603.508,A -85,B 0,C 180,E1 -14466.161,E2 -14466.161} C_VEL
LIN {X 0,Y 343.75,Z 672.83,A -85,B 0,C 180,E1 -14468.208,E2 -14468.208} C_VEL
LIN {X 0,Y 342.784,Z 685.965,A -85,B 0,C 180,E1 -14468.814,E2 -14468.814} C_VEL
LIN {X 0,Y 341.301,Z 699.338,A -85,B 0,C 180,E1 -14469.664,E2 -14469.664} C_VEL
LIN {X 0,Y 339.926,Z 711.245,A -85,B 0,C 180,E1 -14470.681,E2 -14470.681} C_VEL
LIN {X 0,Y 338.47,Z 722.119,A -85,B 0,C 180,E1 -14471.851,E2 -14471.851} C_VEL
LIN {X 0,Y 336.809,Z 733.26,A -85,B 0,C 180,E1 -14473.356,E2 -14473.356} C_VEL
LIN {X 0,Y 335.409,Z 742.564,A -85,B 0,C 180,E1 -14474.914,E2 -14474.914} C_VEL
LIN {X 0,Y 334.389,Z 750.812,A -85,B 0,C 180,E1 -14476.631,E2 -14476.631} C_VEL
LIN {X 0,Y 333.352,Z 757.928,A -85,B 0,C 180,E1 -14478.444,E2 -14478.444} C_VEL
LIN {X 0,Y 332.743,Z 763.632,A -85,B 0,C 180,E1 -14480.27,E2 -14480.27} C_VEL
LIN {X 0,Y 332.337,Z 768.089,A -85,B 0,C 180,E1 -14482.097,E2 -14482.097} C_VEL
LIN {X 0,Y 332.147,Z 771.522,A -85,B 0,C 180,E1 -14483.984,E2 -14483.984} C_VEL
LIN {X 0,Y 332.141,Z 773.074,A -85,B 0,C 180,E1 -14485.143,E2 -14485.143} C_VEL
LIN {X 0,Y 332.15,Z 774.26,A -85,B 0,C 180,E1 -14486.359,E2 -14486.359} C_VEL
LIN {X 0,Y 332.199,Z 775.025,A -85,B 0,C 180,E1 -14487.573,E2 -14487.573} C_VEL
LIN {X 0,Y 332.353,Z 775.357,A -85,B 0,C 180,E1 -14488.786,E2 -14488.786} C_VEL
LIN {X 0,Y 332.397,Z 775.197,A -85,B 0,C 180,E1 -14489.998,E2 -14489.998} C_VEL
LIN {X 0,Y 332.375,Z 774.606,A -85,B 0,C 180,E1 -14491.21,E2 -14491.21} C_VEL
LIN {X 0,Y 332.3,Z 773.576,A -85,B 0,C 180,E1 -14492.422,E2 -14492.422} C_VEL
LIN {X 0,Y 332.205,Z 772.034,A -85,B 0,C 180,E1 -14493.637,E2 -14493.637} C_VEL
LIN {X 0,Y 332.302,Z 770.045,A -85,B 0,C 180,E1 -14494.851,E2 -14494.851} C_VEL
LIN {X 0,Y 332.246,Z 766.227,A -85,B 0,C 180,E1 -14496.618,E2 -14496.618} C_VEL
LIN {X 0,Y 332.432,Z 760.872,A -85,B 0,C 180,E1 -14498.508,E2 -14498.508} C_VEL
LIN {X 0,Y 332.762,Z 754.192,A -85,B 0,C 180,E1 -14500.34,E2 -14500.34} C_VEL
LIN {X 0,Y 333.349,Z 745.812,A -85,B 0,C 180,E1 -14502.169,E2 -14502.169} C_VEL
LIN {X 0,Y 334.06,Z 737.202,A -85,B 0,C 180,E1 -14503.688,E2 -14503.688} C_VEL
LIN {X 0,Y 334.749,Z 727.856,A -85,B 0,C 180,E1 -14505.035,E2 -14505.035} C_VEL
LIN {X 0,Y 335.64,Z 717.384,A -85,B 0,C 180,E1 -14506.262,E2 -14506.262} C_VEL
LIN {X 0,Y 336.559,Z 706.197,A -85,B 0,C 180,E1 -14507.309,E2 -14507.309} C_VEL
LIN {X 0,Y 337.429,Z 693.766,A -85,B 0,C 180,E1 -14508.203,E2 -14508.203} C_VEL
LIN {X 0,Y 338.81,Z 677.876,A -85,B 0,C 180,E1 -14509.303,E2 -14509.303} C_VEL
LIN {X 0,Y 339.65,Z 664.389,A -85,B 0,C 180,E1 -14509.961,E2 -14509.961} C_VEL
LIN {X 0,Y 340.113,Z 651.138,A -85,B 0,C 180,E1 -14510.366,E2 -14510.366} C_VEL
LIN {X 0,Y 340.794,Z 598.729,A -85,B 0,C 180,E1 -14511.473,E2 -14511.473} C_VEL
LIN {X 0,Y 336.284,Z 550.628,A -85,B 0,C 180,E1 -14512.8,E2 -14512.8} C_VEL
LIN {X 0,Y 335.96,Z 544.912,A -85,B 0,C 180,E1 -14513.12,E2 -14513.12} C_VEL
LIN {X 0,Y 337.956,Z 523.006,A -85,B 0,C 180,E1 -14517.224,E2 -14517.224} C_VEL
LIN {X 0,Y 339.288,Z 509.357,A -85,B 0,C 180,E1 -14519.808,E2 -14519.808} C_VEL
LIN {X 0,Y 337.138,Z 498.378,A -85,B 0,C 180,E1 -14522.109,E2 -14522.109} C_VEL
LIN {X 0,Y 333.97,Z 484.107,A -85,B 0,C 180,E1 -14525.234,E2 -14525.234} C_VEL
LIN {X 0,Y 333.701,Z 483.029,A -85,B 0,C 180,E1 -14525.536,E2 -14525.536} C_VEL
LIN {X 0,Y 333.594,Z 482.928,A -85,B 0,C 180,E1 -14529.197,E2 -14529.197} C_VEL
LIN {X 0,Y 333.621,Z 482.927,A -85,B 0,C 180,E1 -14532.497,E2 -14532.497} C_VEL
LIN {X 0,Y 333.587,Z 482.932,A -85,B 0,C 180,E1 -14535.953,E2 -14535.953} C_VEL
LIN {X 0,Y 333.633,Z 482.923,A -85,B 0,C 180,E1 -14539.315,E2 -14539.315} C_VEL
LIN {X 0,Y 333.653,Z 482.921,A -85,B 0,C 180,E1 -14543.167,E2 -14543.167} C_VEL
LIN {X 0,Y 333.663,Z 482.917,A -85,B 0,C 180,E1 -14545.34,E2 -14545.34} C_VEL
LIN {X 0,Y 333.693,Z 482.916,A -85,B 0,C 180,E1 -14549.708,E2 -14549.708} C_VEL
LIN {X 0,Y 333.723,Z 482.911,A -85,B 0,C 180,E1 -14553.752,E2 -14553.752} C_VEL
LIN {X 0,Y 333.708,Z 482.915,A -85,B 0,C 180,E1 -14557.913,E2 -14557.913} C_VEL
LIN {X 0,Y 333.781,Z 482.903,A -85,B 0,C 180,E1 -14561.588,E2 -14561.588} C_VEL
LIN {X 0,Y 333.795,Z 482.903,A -85,B 0,C 180,E1 -14565.576,E2 -14565.576} C_VEL
LIN {X 0,Y 333.821,Z 482.897,A -85,B 0,C 180,E1 -14569.077,E2 -14569.077} C_VEL
LIN {X 0,Y 334.011,Z 482.879,A -85,B 0,C 180,E1 -14572.747,E2 -14572.747} C_VEL
LIN {X 0,Y 333.795,Z 482.903,A -85,B 0,C 180,E1 -14575.168,E2 -14575.168} C_VEL
LIN {X 0,Y 334.091,Z 482.863,A -85,B 0,C 180,E1 -14577.588,E2 -14577.588} C_VEL
LIN {X 0,Y 334.233,Z 482.846,A -85,B 0,C 180,E1 -14580,E2 -14580} C_VEL
LIN {X 0,Y 334.092,Z 482.869,A -85,B 0,C 180,E1 -14582.411,E2 -14582.411} C_VEL
LIN {X 0,Y 334.01,Z 482.874,A -85,B 0,C 180,E1 -14587.252,E2 -14587.252} C_VEL
LIN {X 0,Y 333.82,Z 482.902,A -85,B 0,C 180,E1 -14590.922,E2 -14590.922} C_VEL
LIN {X 0,Y 333.794,Z 482.909,A -85,B 0,C 180,E1 -14594.634,E2 -14594.634} C_VEL
LIN {X 0,Y 333.783,Z 482.906,A -85,B 0,C 180,E1 -14598.656,E2 -14598.656} C_VEL
LIN {X 0,Y 333.678,Z 482.918,A -85,B 0,C 180,E1 -14602.279,E2 -14602.279} C_VEL
LIN {X 0,Y 333.722,Z 482.913,A -85,B 0,C 180,E1 -14606.247,E2 -14606.247} C_VEL
LIN {X 0,Y 333.697,Z 482.916,A -85,B 0,C 180,E1 -14608.973,E2 -14608.973} C_VEL
LIN {X 0,Y 333.63,Z 482.927,A -85,B 0,C 180,E1 -14612.588,E2 -14612.588} C_VEL
LIN {X 0,Y 333.664,Z 482.919,A -85,B 0,C 180,E1 -14616.14,E2 -14616.14} C_VEL
LIN {X 0,Y 333.634,Z 482.925,A -85,B 0,C 180,E1 -14619.193,E2 -14619.193} C_VEL
LIN {X 0,Y 333.622,Z 482.927,A -85,B 0,C 180,E1 -14622.502,E2 -14622.502} C_VEL
LIN {X 0,Y 333.658,Z 482.919,A -85,B 0,C 180,E1 -14625.968,E2 -14625.968} C_VEL
LIN {X 0,Y 333.691,Z 482.917,A -85,B 0,C 180,E1 -14629.306,E2 -14629.306} C_VEL
LIN {X 0,Y 333.659,Z 482.917,A -85,B 0,C 180,E1 -14633.168,E2 -14633.168} C_VEL
LIN {X 0,Y 333.627,Z 482.926,A -85,B 0,C 180,E1 -14636.793,E2 -14636.793} C_VEL
LIN {X 0,Y 333.694,Z 482.915,A -85,B 0,C 180,E1 -14639.712,E2 -14639.712} C_VEL
LIN {X 0,Y 333.734,Z 482.907,A -85,B 0,C 180,E1 -14642.403,E2 -14642.403} C_VEL
LIN {X 0,Y 333.72,Z 482.918,A -85,B 0,C 180,E1 -14645.093,E2 -14645.093} C_VEL
LIN {X 0,Y 333.674,Z 482.921,A -85,B 0,C 180,E1 -14649.021,E2 -14649.021} C_VEL
LIN {X 0,Y 333.788,Z 482.905,A -85,B 0,C 180,E1 -14651.591,E2 -14651.591} C_VEL
LIN {X 0,Y 333.803,Z 482.903,A -85,B 0,C 180,E1 -14655.578,E2 -14655.578} C_VEL
LIN {X 0,Y 333.83,Z 482.902,A -85,B 0,C 180,E1 -14659.08,E2 -14659.08} C_VEL
LIN {X 0,Y 334.002,Z 482.976,A -85,B 0,C 180,E1 -14661.675,E2 -14661.675} C_VEL
LIN {X 0,Y 334.179,Z 483.804,A -85,B 0,C 180,E1 -14661.894,E2 -14661.894} C_VEL
LIN {X 0,Y 341.004,Z 502.253,A -85,B 0,C 180,E1 -14662.721,E2 -14662.721} C_VEL
LIN {X 0,Y 341.893,Z 505.588,A -85,B 0,C 180,E1 -14662.843,E2 -14662.843} C_VEL
LIN {X 0,Y 341.091,Z 558.565,A -85,B 0,C 180,E1 -14663.959,E2 -14663.959} C_VEL
LIN {X 0,Y 341.042,Z 571.607,A -85,B 0,C 180,E1 -14664.348,E2 -14664.348} C_VEL
LIN {X 0,Y 340.767,Z 584.485,A -85,B 0,C 180,E1 -14664.973,E2 -14664.973} C_VEL
LIN {X 0,Y 340.229,Z 597.386,A -85,B 0,C 180,E1 -14665.856,E2 -14665.856} C_VEL
LIN {X 0,Y 339.543,Z 608.689,A -85,B 0,C 180,E1 -14666.887,E2 -14666.887} C_VEL
LIN {X 0,Y 338.643,Z 620.16,A -85,B 0,C 180,E1 -14668.218,E2 -14668.218} C_VEL
LIN {X 0,Y 337.786,Z 630.129,A -85,B 0,C 180,E1 -14669.669,E2 -14669.669} C_VEL
LIN {X 0,Y 336.897,Z 638.628,A -85,B 0,C 180,E1 -14671.197,E2 -14671.197} C_VEL
LIN {X 0,Y 336.067,Z 646.734,A -85,B 0,C 180,E1 -14672.999,E2 -14672.999} C_VEL
LIN {X 0,Y 335.36,Z 653.28,A -85,B 0,C 180,E1 -14674.811,E2 -14674.811} C_VEL
LIN {X 0,Y 334.835,Z 658.499,A -85,B 0,C 180,E1 -14676.631,E2 -14676.631} C_VEL
LIN {X 0,Y 334.293,Z 663.283,A -85,B 0,C 180,E1 -14678.85,E2 -14678.85} C_VEL
LIN {X 0,Y 334.008,Z 666.384,A -85,B 0,C 180,E1 -14680.918,E2 -14680.918} C_VEL
LIN {X 0,Y 333.93,Z 667.67,A -85,B 0,C 180,E1 -14682.151,E2 -14682.151} C_VEL
LIN {X 0,Y 333.928,Z 668.528,A -85,B 0,C 180,E1 -14683.388,E2 -14683.388} C_VEL
LIN {X 0,Y 334.003,Z 668.96,A -85,B 0,C 180,E1 -14684.628,E2 -14684.628} C_VEL
LIN {X 0,Y 334.138,Z 669.006,A -85,B 0,C 180,E1 -14685.871,E2 -14685.871} C_VEL
LIN {X 0,Y 334.299,Z 668.663,A -85,B 0,C 180,E1 -14687.119,E2 -14687.119} C_VEL
LIN {X 0,Y 334.828,Z 667.132,A -85,B 0,C 180,E1 -14689.172,E2 -14689.172} C_VEL
LIN {X 0,Y 335.615,Z 663.969,A -85,B 0,C 180,E1 -14691.5,E2 -14691.5} C_VEL
LIN {X 0,Y 336.479,Z 660.213,A -85,B 0,C 180,E1 -14693.383,E2 -14693.383} C_VEL
LIN {X 0,Y 337.543,Z 655.241,A -85,B 0,C 180,E1 -14695.269,E2 -14695.269} C_VEL
LIN {X 0,Y 338.834,Z 648.863,A -85,B 0,C 180,E1 -14697.152,E2 -14697.152} C_VEL
LIN {X 0,Y 340.285,Z 640.716,A -85,B 0,C 180,E1 -14699.038,E2 -14699.038} C_VEL
LIN {X 0,Y 341.742,Z 632.081,A -85,B 0,C 180,E1 -14700.635,E2 -14700.635} C_VEL
LIN {X 0,Y 342.967,Z 622.927,A -85,B 0,C 180,E1 -14702.023,E2 -14702.023} C_VEL
LIN {X 0,Y 344.321,Z 612.387,A -85,B 0,C 180,E1 -14703.289,E2 -14703.289} C_VEL
LIN {X 0,Y 345.416,Z 601.037,A -85,B 0,C 180,E1 -14704.378,E2 -14704.378} C_VEL
LIN {X 0,Y 346.252,Z 588.721,A -85,B 0,C 180,E1 -14705.288,E2 -14705.288} C_VEL
LIN {X 0,Y 346.758,Z 575.716,A -85,B 0,C 180,E1 -14705.972,E2 -14705.972} C_VEL
LIN {X 0,Y 346.9,Z 563.44,A -85,B 0,C 180,E1 -14706.397,E2 -14706.397} C_VEL
LIN {X 0,Y 347.04,Z 546.301,A -85,B 0,C 180,E1 -14706.788,E2 -14706.788} C_VEL
LIN {X 0,Y 346.587,Z 540.506,A -85,B 0,C 180,E1 -14706.962,E2 -14706.962} C_VEL
LIN {X 0,Y 341.971,Z 521.909,A -85,B 0,C 180,E1 -14707.816,E2 -14707.816} C_VEL
LIN {X 0,Y 341.534,Z 516.115,A -85,B 0,C 180,E1 -14707.994,E2 -14707.994} C_VEL
LIN {X 0,Y 341.451,Z 513.34,A -85,B 0,C 180,E1 -14708.068,E2 -14708.068} C_VEL
LIN {X 0,Y 333.079,Z 496.394,A -85,B 0,C 180,E1 -14709.299,E2 -14709.299} C_VEL
LIN {X 0,Y 327.609,Z 486.611,A -85,B 0,C 180,E1 -14710.115,E2 -14710.115} C_VEL
LIN {X 0,Y 326.739,Z 484.487,A -85,B 0,C 180,E1 -14710.335,E2 -14710.335} C_VEL
LIN {X 0,Y 326.626,Z 483.845,A -85,B 0,C 180,E1 -14710.61,E2 -14710.61} C_VEL
LIN {X 0,Y 326.567,Z 483.802,A -85,B 0,C 180,E1 -14713.527,E2 -14713.527} C_VEL
LIN {X 0,Y 326.612,Z 484.022,A -85,B 0,C 180,E1 -14715.903,E2 -14715.903} C_VEL
LIN {X 0,Y 330.098,Z 498.987,A -85,B 0,C 180,E1 -14719.114,E2 -14719.114} C_VEL
LIN {X 0,Y 332.058,Z 508.673,A -85,B 0,C 180,E1 -14721.137,E2 -14721.137} C_VEL
LIN {X 0,Y 331.248,Z 525.133,A -85,B 0,C 180,E1 -14724.215,E2 -14724.215} C_VEL
LIN {X 0,Y 334.785,Z 549.14,A -85,B 0,C 180,E1 -14725.102,E2 -14725.102} C_VEL
LIN {X 0,Y 332.232,Z 636.499,A -85,B 0,C 180,E1 -14727.492,E2 -14727.492} C_VEL
LIN {X 0,Y 331.599,Z 649.839,A -85,B 0,C 180,E1 -14728.094,E2 -14728.094} C_VEL
LIN {X 0,Y 330.829,Z 663.572,A -85,B 0,C 180,E1 -14728.993,E2 -14728.993} C_VEL
LIN {X 0,Y 330.082,Z 674.901,A -85,B 0,C 180,E1 -14729.977,E2 -14729.977} C_VEL
LIN {X 0,Y 329.19,Z 685.924,A -85,B 0,C 180,E1 -14731.181,E2 -14731.181} C_VEL
LIN {X 0,Y 328.277,Z 696.394,A -85,B 0,C 180,E1 -14732.595,E2 -14732.595} C_VEL
LIN {X 0,Y 327.386,Z 706.192,A -85,B 0,C 180,E1 -14734.242,E2 -14734.242} C_VEL
LIN {X 0,Y 326.697,Z 714.134,A -85,B 0,C 180,E1 -14735.875,E2 -14735.875} C_VEL
LIN {X 0,Y 326.112,Z 721.19,A -85,B 0,C 180,E1 -14737.654,E2 -14737.654} C_VEL
LIN {X 0,Y 325.563,Z 727.837,A -85,B 0,C 180,E1 -14739.795,E2 -14739.795} C_VEL
LIN {X 0,Y 325.223,Z 732.913,A -85,B 0,C 180,E1 -14741.963,E2 -14741.963} C_VEL
LIN {X 0,Y 324.991,Z 735.822,A -85,B 0,C 180,E1 -14743.673,E2 -14743.673} C_VEL
LIN {X 0,Y 324.933,Z 737.425,A -85,B 0,C 180,E1 -14744.957,E2 -14744.957} C_VEL
LIN {X 0,Y 325.002,Z 738.869,A -85,B 0,C 180,E1 -14746.687,E2 -14746.687} C_VEL
LIN {X 0,Y 325.051,Z 739.477,A -85,B 0,C 180,E1 -14748.78,E2 -14748.78} C_VEL
LIN {X 0,Y 325.191,Z 739.258,A -85,B 0,C 180,E1 -14750.044,E2 -14750.044} C_VEL
LIN {X 0,Y 325.407,Z 738.619,A -85,B 0,C 180,E1 -14751.305,E2 -14751.305} C_VEL
LIN {X 0,Y 325.784,Z 737.103,A -85,B 0,C 180,E1 -14752.916,E2 -14752.916} C_VEL
LIN {X 0,Y 326.397,Z 733.965,A -85,B 0,C 180,E1 -14755.06,E2 -14755.06} C_VEL
LIN {X 0,Y 327.08,Z 730.084,A -85,B 0,C 180,E1 -14756.921,E2 -14756.921} C_VEL
LIN {X 0,Y 328.098,Z 724.987,A -85,B 0,C 180,E1 -14758.773,E2 -14758.773} C_VEL
LIN {X 0,Y 329.305,Z 718.567,A -85,B 0,C 180,E1 -14760.612,E2 -14760.612} C_VEL
LIN {X 0,Y 330.839,Z 710.564,A -85,B 0,C 180,E1 -14762.435,E2 -14762.435} C_VEL
LIN {X 0,Y 332.223,Z 702.376,A -85,B 0,C 180,E1 -14763.943,E2 -14763.943} C_VEL
LIN {X 0,Y 334.008,Z 691.344,A -85,B 0,C 180,E1 -14765.585,E2 -14765.585} C_VEL
LIN {X 0,Y 335.583,Z 680.02,A -85,B 0,C 180,E1 -14766.917,E2 -14766.917} C_VEL
LIN {X 0,Y 336.916,Z 668.983,A -85,B 0,C 180,E1 -14767.944,E2 -14767.944} C_VEL
LIN {X 0,Y 338.148,Z 656.867,A -85,B 0,C 180,E1 -14768.818,E2 -14768.818} C_VEL
LIN {X 0,Y 339.069,Z 643.827,A -85,B 0,C 180,E1 -14769.508,E2 -14769.508} C_VEL
LIN {X 0,Y 339.873,Z 628.157,A -85,B 0,C 180,E1 -14770.048,E2 -14770.048} C_VEL
LIN {X 0,Y 344.045,Z 553.836,A -85,B 0,C 180,E1 -14772.279,E2 -14772.279} C_VEL
LIN {X 0,Y 341.264,Z 539.72,A -85,B 0,C 180,E1 -14773.198,E2 -14773.198} C_VEL
LIN {X 0,Y 338.878,Z 529.621,A -85,B 0,C 180,E1 -14773.997,E2 -14773.997} C_VEL
LIN {X 0,Y 339.375,Z 524.486,A -85,B 0,C 180,E1 -14775.003,E2 -14775.003} C_VEL
LIN {X 0,Y 338.079,Z 516.363,A -85,B 0,C 180,E1 -14777.006,E2 -14777.006} C_VEL
LIN {X 0,Y 335.999,Z 507.942,A -85,B 0,C 180,E1 -14779.313,E2 -14779.313} C_VEL
LIN {X 0,Y 333.582,Z 500.47,A -85,B 0,C 180,E1 -14781.619,E2 -14781.619} C_VEL
LIN {X 0,Y 330.289,Z 492.024,A -85,B 0,C 180,E1 -14784.515,E2 -14784.515} C_VEL
LIN {X 0,Y 328.609,Z 488.066,A -85,B 0,C 180,E1 -14786.066,E2 -14786.066} C_VEL
LIN {X 0,Y 326.733,Z 484.146,A -85,B 0,C 180,E1 -14787.862,E2 -14787.862} C_VEL
LIN {X 0,Y 326.676,Z 483.848,A -85,B 0,C 180,E1 -14788.249,E2 -14788.249} C_VEL
LIN {X 0,Y 326.599,Z 483.805,A -85,B 0,C 180,E1 -14791.095,E2 -14791.095} C_VEL
LIN {X 0,Y 326.616,Z 483.797,A -85,B 0,C 180,E1 -14794.019,E2 -14794.019} C_VEL
LIN {X 0,Y 326.636,Z 483.799,A -85,B 0,C 180,E1 -14797.238,E2 -14797.238} C_VEL
LIN {X 0,Y 326.587,Z 483.806,A -85,B 0,C 180,E1 -14801.131,E2 -14801.131} C_VEL
LIN {X 0,Y 326.536,Z 483.808,A -85,B 0,C 180,E1 -14804.742,E2 -14804.742} C_VEL
LIN {X 0,Y 326.584,Z 483.802,A -85,B 0,C 180,E1 -14808.153,E2 -14808.153} C_VEL
LIN {X 0,Y 326.652,Z 484.043,A -85,B 0,C 180,E1 -14810.338,E2 -14810.338} C_VEL
LIN {X 0,Y 330.067,Z 495.868,A -85,B 0,C 180,E1 -14813.65,E2 -14813.65} C_VEL
LIN {X 0,Y 333.24,Z 508.964,A -85,B 0,C 180,E1 -14816.966,E2 -14816.966} C_VEL
LIN {X 0,Y 334.926,Z 517.573,A -85,B 0,C 180,E1 -14819.006,E2 -14819.006} C_VEL
LIN {X 0,Y 334.373,Z 522.602,A -85,B 0,C 180,E1 -14819.965,E2 -14819.965} C_VEL
LIN {X 0,Y 335.505,Z 538.083,A -85,B 0,C 180,E1 -14821.619,E2 -14821.619} C_VEL
LIN {X 0,Y 336.62,Z 551.655,A -85,B 0,C 180,E1 -14822.862,E2 -14822.862} C_VEL
LIN {X 0,Y 338.977,Z 568.132,A -85,B 0,C 180,E1 -14823.857,E2 -14823.857} C_VEL
LIN {X 0,Y 340.45,Z 583.756,A -85,B 0,C 180,E1 -14824.65,E2 -14824.65} C_VEL
LIN {X 0,Y 341.296,Z 603.603,A -85,B 0,C 180,E1 -14825.5,E2 -14825.5} C_VEL
LIN {X 0,Y 337.571,Z 673.234,A -85,B 0,C 180,E1 -14827.627,E2 -14827.627} C_VEL
LIN {X 0,Y 336.39,Z 687.351,A -85,B 0,C 180,E1 -14828.311,E2 -14828.311} C_VEL
LIN {X 0,Y 334.77,Z 701.057,A -85,B 0,C 180,E1 -14829.25,E2 -14829.25} C_VEL
LIN {X 0,Y 333.326,Z 712.396,A -85,B 0,C 180,E1 -14830.282,E2 -14830.282} C_VEL
LIN {X 0,Y 331.417,Z 725.236,A -85,B 0,C 180,E1 -14831.771,E2 -14831.771} C_VEL
LIN {X 0,Y 329.874,Z 734.871,A -85,B 0,C 180,E1 -14833.171,E2 -14833.171} C_VEL
LIN {X 0,Y 328.387,Z 744.325,A -85,B 0,C 180,E1 -14834.874,E2 -14834.874} C_VEL
LIN {X 0,Y 327.288,Z 752.301,A -85,B 0,C 180,E1 -14836.652,E2 -14836.652} C_VEL
LIN {X 0,Y 326.358,Z 757.98,A -85,B 0,C 180,E1 -14838.193,E2 -14838.193} C_VEL
LIN {X 0,Y 325.728,Z 763.59,A -85,B 0,C 180,E1 -14840.058,E2 -14840.058} C_VEL
LIN {X 0,Y 325.265,Z 767.96,A -85,B 0,C 180,E1 -14841.924,E2 -14841.924} C_VEL
LIN {X 0,Y 325.059,Z 771.526,A -85,B 0,C 180,E1 -14844.021,E2 -14844.021} C_VEL
LIN {X 0,Y 325.07,Z 773.935,A -85,B 0,C 180,E1 -14846.279,E2 -14846.279} C_VEL
LIN {X 0,Y 325.102,Z 774.663,A -85,B 0,C 180,E1 -14847.52,E2 -14847.52} C_VEL
LIN {X 0,Y 325.268,Z 774.922,A -85,B 0,C 180,E1 -14848.76,E2 -14848.76} C_VEL
LIN {X 0,Y 325.332,Z 774.727,A -85,B 0,C 180,E1 -14849.998,E2 -14849.998} C_VEL
LIN {X 0,Y 325.311,Z 774.097,A -85,B 0,C 180,E1 -14851.236,E2 -14851.236} C_VEL
LIN {X 0,Y 325.207,Z 772.994,A -85,B 0,C 180,E1 -14852.475,E2 -14852.475} C_VEL
LIN {X 0,Y 325.173,Z 770.453,A -85,B 0,C 180,E1 -14854.336,E2 -14854.336} C_VEL
LIN {X 0,Y 325.193,Z 766.782,A -85,B 0,C 180,E1 -14856.201,E2 -14856.201} C_VEL
LIN {X 0,Y 325.298,Z 761.871,A -85,B 0,C 180,E1 -14858.071,E2 -14858.071} C_VEL
LIN {X 0,Y 325.589,Z 755.583,A -85,B 0,C 180,E1 -14859.942,E2 -14859.942} C_VEL
LIN {X 0,Y 326.104,Z 747.67,A -85,B 0,C 180,E1 -14861.812,E2 -14861.812} C_VEL
LIN {X 0,Y 326.691,Z 739.482,A -85,B 0,C 180,E1 -14863.369,E2 -14863.369} C_VEL
LIN {X 0,Y 327.395,Z 731.676,A -85,B 0,C 180,E1 -14864.607,E2 -14864.607} C_VEL
LIN {X 0,Y 328.317,Z 721.162,A -85,B 0,C 180,E1 -14865.98,E2 -14865.98} C_VEL
LIN {X 0,Y 329.188,Z 710.826,A -85,B 0,C 180,E1 -14867.069,E2 -14867.069} C_VEL
LIN {X 0,Y 330.06,Z 698.798,A -85,B 0,C 180,E1 -14868.062,E2 -14868.062} C_VEL
LIN {X 0,Y 330.822,Z 689.428,A -85,B 0,C 180,E1 -14868.74,E2 -14868.74} C_VEL
LIN {X 0,Y 331.943,Z 676.75,A -85,B 0,C 180,E1 -14869.638,E2 -14869.638} C_VEL
LIN {X 0,Y 332.785,Z 664.138,A -85,B 0,C 180,E1 -14870.27,E2 -14870.27} C_VEL
LIN {X 0,Y 333.281,Z 651.365,A -85,B 0,C 180,E1 -14870.682,E2 -14870.682} C_VEL
LIN {X 0,Y 334.09,Z 600.209,A -85,B 0,C 180,E1 -14871.783,E2 -14871.783} C_VEL
LIN {X 0,Y 329.294,Z 549.111,A -85,B 0,C 180,E1 -14873.227,E2 -14873.227} C_VEL
LIN {X 0,Y 329.05,Z 543.859,A -85,B 0,C 180,E1 -14873.548,E2 -14873.548} C_VEL
LIN {X 0,Y 331.221,Z 521.562,A -85,B 0,C 180,E1 -14877.825,E2 -14877.825} C_VEL
LIN {X 0,Y 332.318,Z 510.956,A -85,B 0,C 180,E1 -14879.877,E2 -14879.877} C_VEL
LIN {X 0,Y 330.72,Z 501.977,A -85,B 0,C 180,E1 -14881.785,E2 -14881.785} C_VEL
LIN {X 0,Y 327.222,Z 486.234,A -85,B 0,C 180,E1 -14885.297,E2 -14885.297} C_VEL
LIN {X 0,Y 326.669,Z 483.914,A -85,B 0,C 180,E1 -14885.889,E2 -14885.889} C_VEL
LIN {X 0,Y 326.564,Z 483.804,A -85,B 0,C 180,E1 -14889.216,E2 -14889.216} C_VEL
LIN {X 0,Y 326.566,Z 483.804,A -85,B 0,C 180,E1 -14892.969,E2 -14892.969} C_VEL
LIN {X 0,Y 326.566,Z 483.804,A -85,B 0,C 180,E1 -14897.026,E2 -14897.026} C_VEL
LIN {X 0,Y 326.589,Z 483.802,A -85,B 0,C 180,E1 -14900.774,E2 -14900.774} C_VEL
LIN {X 0,Y 326.602,Z 483.8,A -85,B 0,C 180,E1 -14904.478,E2 -14904.478} C_VEL
LIN {X 0,Y 326.597,Z 483.799,A -85,B 0,C 180,E1 -14907.454,E2 -14907.454} C_VEL
LIN {X 0,Y 326.65,Z 483.796,A -85,B 0,C 180,E1 -14910.339,E2 -14910.339} C_VEL
LIN {X 0,Y 326.678,Z 483.794,A -85,B 0,C 180,E1 -14914.515,E2 -14914.515} C_VEL
LIN {X 0,Y 326.633,Z 483.797,A -85,B 0,C 180,E1 -14918.544,E2 -14918.544} C_VEL
LIN {X 0,Y 326.732,Z 483.781,A -85,B 0,C 180,E1 -14921.176,E2 -14921.176} C_VEL
LIN {X 0,Y 326.75,Z 483.78,A -85,B 0,C 180,E1 -14925.432,E2 -14925.432} C_VEL
LIN {X 0,Y 326.757,Z 483.778,A -85,B 0,C 180,E1 -14928.838,E2 -14928.838} C_VEL
LIN {X 0,Y 326.965,Z 483.759,A -85,B 0,C 180,E1 -14932.59,E2 -14932.59} C_VEL
LIN {X 0,Y 326.762,Z 483.779,A -85,B 0,C 180,E1 -14935.064,E2 -14935.064} C_VEL
LIN {X 0,Y 327.032,Z 483.742,A -85,B 0,C 180,E1 -14937.536,E2 -14937.536} C_VEL
LIN {X 0,Y 327.184,Z 483.723,A -85,B 0,C 180,E1 -14940,E2 -14940} C_VEL
LIN {X 0,Y 327.033,Z 483.749,A -85,B 0,C 180,E1 -14942.463,E2 -14942.463} C_VEL
LIN {X 0,Y 326.955,Z 483.752,A -85,B 0,C 180,E1 -14946.723,E2 -14946.723} C_VEL
LIN {X 0,Y 326.8,Z 483.77,A -85,B 0,C 180,E1 -14949.906,E2 -14949.906} C_VEL
LIN {X 0,Y 326.745,Z 483.781,A -85,B 0,C 180,E1 -14953.686,E2 -14953.686} C_VEL
LIN {X 0,Y 326.685,Z 483.786,A -85,B 0,C 180,E1 -14957.528,E2 -14957.528} C_VEL
LIN {X 0,Y 326.651,Z 483.789,A -85,B 0,C 180,E1 -14960.135,E2 -14960.135} C_VEL
LIN {X 0,Y 326.638,Z 483.795,A -85,B 0,C 180,E1 -14964.129,E2 -14964.129} C_VEL
LIN {X 0,Y 326.671,Z 483.792,A -85,B 0,C 180,E1 -14966.858,E2 -14966.858} C_VEL
LIN {X 0,Y 326.626,Z 483.797,A -85,B 0,C 180,E1 -14970.612,E2 -14970.612} C_VEL
LIN {X 0,Y 326.594,Z 483.8,A -85,B 0,C 180,E1 -14974.02,E2 -14974.02} C_VEL
LIN {X 0,Y 326.615,Z 483.796,A -85,B 0,C 180,E1 -14977.24,E2 -14977.24} C_VEL
LIN {X 0,Y 326.566,Z 483.807,A -85,B 0,C 180,E1 -14981.133,E2 -14981.133} C_VEL
LIN {X 0,Y 326.571,Z 483.805,A -85,B 0,C 180,E1 -14984.754,E2 -14984.754} C_VEL
LIN {X 0,Y 326.612,Z 483.798,A -85,B 0,C 180,E1 -14988.163,E2 -14988.163} C_VEL
LIN {X 0,Y 326.641,Z 483.791,A -85,B 0,C 180,E1 -14991.397,E2 -14991.397} C_VEL
LIN {X 0,Y 326.611,Z 483.795,A -85,B 0,C 180,E1 -14994.853,E2 -14994.853} C_VEL
LIN {X 0,Y 326.599,Z 483.801,A -85,B 0,C 180,E1 -14997.457,E2 -14997.457} C_VEL
LIN {X 0,Y 326.652,Z 483.792,A -85,B 0,C 180,E1 -15000.343,E2 -15000.343} C_VEL
LIN {X 0,Y 326.683,Z 483.789,A -85,B 0,C 180,E1 -15004.518,E2 -15004.518} C_VEL
LIN {X 0,Y 326.639,Z 483.793,A -85,B 0,C 180,E1 -15008.547,E2 -15008.547} C_VEL
LIN {X 0,Y 326.739,Z 483.787,A -85,B 0,C 180,E1 -15011.18,E2 -15011.18} C_VEL
LIN {X 0,Y 326.758,Z 483.781,A -85,B 0,C 180,E1 -15015.435,E2 -15015.435} C_VEL
LIN {X 0,Y 326.766,Z 483.782,A -85,B 0,C 180,E1 -15018.841,E2 -15018.841} C_VEL
LIN {X 0,Y 326.929,Z 483.865,A -85,B 0,C 180,E1 -15021.27,E2 -15021.27} C_VEL
LIN {X 0,Y 327.143,Z 484.775,A -85,B 0,C 180,E1 -15021.498,E2 -15021.498} C_VEL
LIN {X 0,Y 334.23,Z 503.607,A -85,B 0,C 180,E1 -15022.366,E2 -15022.366} C_VEL
LIN {X 0,Y 335.125,Z 506.756,A -85,B 0,C 180,E1 -15022.489,E2 -15022.489} C_VEL
LIN {X 0,Y 334.319,Z 558.998,A -85,B 0,C 180,E1 -15023.612,E2 -15023.612} C_VEL
LIN {X 0,Y 334.279,Z 572.211,A -85,B 0,C 180,E1 -15024.006,E2 -15024.006} C_VEL
LIN {X 0,Y 333.969,Z 585.204,A -85,B 0,C 180,E1 -15024.644,E2 -15024.644} C_VEL
LIN {X 0,Y 333.471,Z 597.19,A -85,B 0,C 180,E1 -15025.469,E2 -15025.469} C_VEL
LIN {X 0,Y 332.766,Z 608.81,A -85,B 0,C 180,E1 -15026.521,E2 -15026.521} C_VEL
LIN {X 0,Y 331.848,Z 620.424,A -85,B 0,C 180,E1 -15027.878,E2 -15027.878} C_VEL
LIN {X 0,Y 330.93,Z 630.35,A -85,B 0,C 180,E1 -15029.327,E2 -15029.327} C_VEL
LIN {X 0,Y 329.962,Z 639.568,A -85,B 0,C 180,E1 -15031.001,E2 -15031.001} C_VEL
LIN {X 0,Y 329.147,Z 647.343,A -85,B 0,C 180,E1 -15032.756,E2 -15032.756} C_VEL
LIN {X 0,Y 328.489,Z 652.959,A -85,B 0,C 180,E1 -15034.296,E2 -15034.296} C_VEL
LIN {X 0,Y 327.9,Z 658.436,A -85,B 0,C 180,E1 -15036.154,E2 -15036.154} C_VEL
LIN {X 0,Y 327.452,Z 662.744,A -85,B 0,C 180,E1 -15038.021,E2 -15038.021} C_VEL
LIN {X 0,Y 327.091,Z 666.004,A -85,B 0,C 180,E1 -15039.9,E2 -15039.9} C_VEL
LIN {X 0,Y 326.955,Z 667.635,A -85,B 0,C 180,E1 -15041.157,E2 -15041.157} C_VEL
LIN {X 0,Y 326.909,Z 668.842,A -85,B 0,C 180,E1 -15042.417,E2 -15042.417} C_VEL
LIN {X 0,Y 327.005,Z 669.989,A -85,B 0,C 180,E1 -15044.948,E2 -15044.948} C_VEL
LIN {X 0,Y 327.165,Z 669.981,A -85,B 0,C 180,E1 -15046.218,E2 -15046.218} C_VEL
LIN {X 0,Y 327.352,Z 669.535,A -85,B 0,C 180,E1 -15047.494,E2 -15047.494} C_VEL
LIN {X 0,Y 327.891,Z 668.064,A -85,B 0,C 180,E1 -15049.424,E2 -15049.424} C_VEL
LIN {X 0,Y 328.801,Z 664.599,A -85,B 0,C 180,E1 -15051.968,E2 -15051.968} C_VEL
LIN {X 0,Y 329.751,Z 660.714,A -85,B 0,C 180,E1 -15053.89,E2 -15053.89} C_VEL
LIN {X 0,Y 331.134,Z 654.571,A -85,B 0,C 180,E1 -15056.131,E2 -15056.131} C_VEL
LIN {X 0,Y 332.527,Z 647.737,A -85,B 0,C 180,E1 -15058.053,E2 -15058.053} C_VEL
LIN {X 0,Y 333.832,Z 640.654,A -85,B 0,C 180,E1 -15059.654,E2 -15059.654} C_VEL
LIN {X 0,Y 335.338,Z 632.046,A -85,B 0,C 180,E1 -15061.234,E2 -15061.234} C_VEL
LIN {X 0,Y 336.688,Z 622.239,A -85,B 0,C 180,E1 -15062.693,E2 -15062.693} C_VEL
LIN {X 0,Y 338.158,Z 611.059,A -85,B 0,C 180,E1 -15064.008,E2 -15064.008} C_VEL
LIN {X 0,Y 339.278,Z 599.363,A -85,B 0,C 180,E1 -15065.09,E2 -15065.09} C_VEL
LIN {X 0,Y 340.054,Z 587.031,A -85,B 0,C 180,E1 -15065.955,E2 -15065.955} C_VEL
LIN {X 0,Y 340.5,Z 574.099,A -85,B 0,C 180,E1 -15066.606,E2 -15066.606} C_VEL
LIN {X 0,Y 340.638,Z 559.959,A -85,B 0,C 180,E1 -15067.034,E2 -15067.034} C_VEL
LIN {X 0,Y 341.534,Z 516.115,A -85,B 0,C 180,E1 -15067.994,E2 -15067.994} C_VEL
LIN {X 0,Y 340.937,Z 512.494,A -85,B 0,C 180,E1 -15068.137,E2 -15068.137} C_VEL
LIN {X 0,Y 339.348,Z 509.296,A -85,B 0,C 180,E1 -15068.365,E2 -15068.365} C_VEL
LIN {X 0,Y 335.858,Z 505.23,A -85,B 0,C 180,E1 -15068.802,E2 -15068.802} C_VEL
LIN {X 0,Y 327.394,Z 497.965,A -85,B 0,C 180,E1 -15069.847,E2 -15069.847} C_VEL
LIN {X 0,Y 323.943,Z 493.433,A -85,B 0,C 180,E1 -15070.333,E2 -15070.333} C_VEL
LIN {X 0,Y 319.741,Z 485.688,A -85,B 0,C 180,E1 -15071.048,E2 -15071.048} C_VEL
LIN {X 0,Y 319.542,Z 484.75,A -85,B 0,C 180,E1 -15071.34,E2 -15071.34} C_VEL
LIN {X 0,Y 319.494,Z 484.687,A -85,B 0,C 180,E1 -15074.744,E2 -15074.744} C_VEL
LIN {X 0,Y 319.552,Z 484.897,A -85,B 0,C 180,E1 -15075.533,E2 -15075.533} C_VEL
LIN {X 0,Y 322.874,Z 498.965,A -85,B 0,C 180,E1 -15078.616,E2 -15078.616} C_VEL
LIN {X 0,Y 325.223,Z 510.707,A -85,B 0,C 180,E1 -15081.076,E2 -15081.076} C_VEL
LIN {X 0,Y 324.388,Z 525.237,A -85,B 0,C 180,E1 -15083.845,E2 -15083.845} C_VEL
LIN {X 0,Y 327.915,Z 550.379,A -85,B 0,C 180,E1 -15084.801,E2 -15084.801} C_VEL
LIN {X 0,Y 325.306,Z 636.515,A -85,B 0,C 180,E1 -15087.218,E2 -15087.218} C_VEL
LIN {X 0,Y 324.71,Z 649.522,A -85,B 0,C 180,E1 -15087.807,E2 -15087.807} C_VEL
LIN {X 0,Y 323.921,Z 663.197,A -85,B 0,C 180,E1 -15088.711,E2 -15088.711} C_VEL
LIN {X 0,Y 323.081,Z 675.521,A -85,B 0,C 180,E1 -15089.799,E2 -15089.799} C_VEL
LIN {X 0,Y 322.106,Z 687.126,A -85,B 0,C 180,E1 -15091.108,E2 -15091.108} C_VEL
LIN {X 0,Y 321.111,Z 697.955,A -85,B 0,C 180,E1 -15092.638,E2 -15092.638} C_VEL
LIN {X 0,Y 320.229,Z 707.812,A -85,B 0,C 180,E1 -15094.371,E2 -15094.371} C_VEL
LIN {X 0,Y 319.558,Z 715.345,A -85,B 0,C 180,E1 -15095.992,E2 -15095.992} C_VEL
LIN {X 0,Y 318.896,Z 722.832,A -85,B 0,C 180,E1 -15097.997,E2 -15097.997} C_VEL
LIN {X 0,Y 318.431,Z 728.729,A -85,B 0,C 180,E1 -15099.996,E2 -15099.996} C_VEL
LIN {X 0,Y 318.123,Z 733.243,A -85,B 0,C 180,E1 -15101.984,E2 -15101.984} C_VEL
LIN {X 0,Y 317.942,Z 735.52,A -85,B 0,C 180,E1 -15103.301,E2 -15103.301} C_VEL
LIN {X 0,Y 317.845,Z 737.327,A -85,B 0,C 180,E1 -15104.614,E2 -15104.614} C_VEL
LIN {X 0,Y 317.912,Z 739.135,A -85,B 0,C 180,E1 -15106.587,E2 -15106.587} C_VEL
LIN {X 0,Y 317.955,Z 739.893,A -85,B 0,C 180,E1 -15108.526,E2 -15108.526} C_VEL
LIN {X 0,Y 318.08,Z 739.836,A -85,B 0,C 180,E1 -15109.819,E2 -15109.819} C_VEL
LIN {X 0,Y 318.286,Z 739.321,A -85,B 0,C 180,E1 -15111.109,E2 -15111.109} C_VEL
LIN {X 0,Y 318.72,Z 737.903,A -85,B 0,C 180,E1 -15112.89,E2 -15112.89} C_VEL
LIN {X 0,Y 319.322,Z 735.181,A -85,B 0,C 180,E1 -15114.95,E2 -15114.95} C_VEL
LIN {X 0,Y 320.006,Z 731.573,A -85,B 0,C 180,E1 -15116.853,E2 -15116.853} C_VEL
LIN {X 0,Y 321.051,Z 726.783,A -85,B 0,C 180,E1 -15118.746,E2 -15118.746} C_VEL
LIN {X 0,Y 322.27,Z 720.722,A -85,B 0,C 180,E1 -15120.625,E2 -15120.625} C_VEL
LIN {X 0,Y 323.859,Z 713.118,A -85,B 0,C 180,E1 -15122.488,E2 -15122.488} C_VEL
LIN {X 0,Y 325.645,Z 703.719,A -85,B 0,C 180,E1 -15124.332,E2 -15124.332} C_VEL
LIN {X 0,Y 327.489,Z 692.867,A -85,B 0,C 180,E1 -15126.006,E2 -15126.006} C_VEL
LIN {X 0,Y 329.181,Z 681.808,A -85,B 0,C 180,E1 -15127.36,E2 -15127.36} C_VEL
LIN {X 0,Y 330.763,Z 669.386,A -85,B 0,C 180,E1 -15128.554,E2 -15128.554} C_VEL
LIN {X 0,Y 332.067,Z 657.386,A -85,B 0,C 180,E1 -15129.441,E2 -15129.441} C_VEL
LIN {X 0,Y 333.133,Z 643.737,A -85,B 0,C 180,E1 -15130.177,E2 -15130.177} C_VEL
LIN {X 0,Y 334.06,Z 626.772,A -85,B 0,C 180,E1 -15130.761,E2 -15130.761} C_VEL
LIN {X 0,Y 338.384,Z 554.999,A -85,B 0,C 180,E1 -15132.98,E2 -15132.98} C_VEL
LIN {X 0,Y 335.352,Z 539.914,A -85,B 0,C 180,E1 -15134.027,E2 -15134.027} C_VEL
LIN {X 0,Y 333.078,Z 530.299,A -85,B 0,C 180,E1 -15134.824,E2 -15134.824} C_VEL
LIN {X 0,Y 333.328,Z 526.606,A -85,B 0,C 180,E1 -15135.595,E2 -15135.595} C_VEL
LIN {X 0,Y 331.578,Z 516.902,A -85,B 0,C 180,E1 -15138.121,E2 -15138.121} C_VEL
LIN {X 0,Y 329.33,Z 508.43,A -85,B 0,C 180,E1 -15140.617,E2 -15140.617} C_VEL
LIN {X 0,Y 326.224,Z 499.693,A -85,B 0,C 180,E1 -15143.606,E2 -15143.606} C_VEL
LIN {X 0,Y 323.588,Z 493.009,A -85,B 0,C 180,E1 -15146.244,E2 -15146.244} C_VEL
LIN {X 0,Y 321.734,Z 489.001,A -85,B 0,C 180,E1 -15148.089,E2 -15148.089} C_VEL
LIN {X 0,Y 319.8,Z 485.682,A -85,B 0,C 180,E1 -15149.998,E2 -15149.998} C_VEL
LIN {X 0,Y 319.615,Z 484.77,A -85,B 0,C 180,E1 -15150.658,E2 -15150.658} C_VEL
LIN {X 0,Y 319.586,Z 484.675,A -85,B 0,C 180,E1 -15153.352,E2 -15153.352} C_VEL
LIN {X 0,Y 319.568,Z 484.676,A -85,B 0,C 180,E1 -15156.427,E2 -15156.427} C_VEL
LIN {X 0,Y 319.568,Z 484.676,A -85,B 0,C 180,E1 -15159.668,E2 -15159.668} C_VEL
LIN {X 0,Y 319.53,Z 484.684,A -85,B 0,C 180,E1 -15163.46,E2 -15163.46} C_VEL
LIN {X 0,Y 319.563,Z 484.678,A -85,B 0,C 180,E1 -15167.016,E2 -15167.016} C_VEL
LIN {X 0,Y 319.571,Z 484.835,A -85,B 0,C 180,E1 -15169.55,E2 -15169.55} C_VEL
LIN {X 0,Y 321.795,Z 492.414,A -85,B 0,C 180,E1 -15171.836,E2 -15171.836} C_VEL
LIN {X 0,Y 324.447,Z 502.235,A -85,B 0,C 180,E1 -15174.523,E2 -15174.523} C_VEL
LIN {X 0,Y 327.288,Z 514.515,A -85,B 0,C 180,E1 -15177.621,E2 -15177.621} C_VEL
LIN {X 0,Y 328.456,Z 519.224,A -85,B 0,C 180,E1 -15178.481,E2 -15178.481} C_VEL
LIN {X 0,Y 329.086,Z 525.346,A -85,B 0,C 180,E1 -15179.297,E2 -15179.297} C_VEL
LIN {X 0,Y 330.233,Z 543.581,A -85,B 0,C 180,E1 -15181.281,E2 -15181.281} C_VEL
LIN {X 0,Y 330.817,Z 551.143,A -85,B 0,C 180,E1 -15181.973,E2 -15181.973} C_VEL
LIN {X 0,Y 333.312,Z 568.842,A -85,B 0,C 180,E1 -15183.104,E2 -15183.104} C_VEL
LIN {X 0,Y 334.735,Z 584.841,A -85,B 0,C 180,E1 -15183.959,E2 -15183.959} C_VEL
LIN {X 0,Y 335.469,Z 604.157,A -85,B 0,C 180,E1 -15184.823,E2 -15184.823} C_VEL
LIN {X 0,Y 331.584,Z 672.046,A -85,B 0,C 180,E1 -15186.953,E2 -15186.953} C_VEL
LIN {X 0,Y 330.489,Z 684.885,A -85,B 0,C 180,E1 -15187.575,E2 -15187.575} C_VEL
LIN {X 0,Y 328.967,Z 697.223,A -85,B 0,C 180,E1 -15188.373,E2 -15188.373} C_VEL
LIN {X 0,Y 327.374,Z 709.238,A -85,B 0,C 180,E1 -15189.417,E2 -15189.417} C_VEL
LIN {X 0,Y 325.72,Z 720.251,A -85,B 0,C 180,E1 -15190.623,E2 -15190.623} C_VEL
LIN {X 0,Y 323.991,Z 730.325,A -85,B 0,C 180,E1 -15191.992,E2 -15191.992} C_VEL
LIN {X 0,Y 322.205,Z 740.828,A -85,B 0,C 180,E1 -15193.778,E2 -15193.778} C_VEL
LIN {X 0,Y 320.909,Z 748.648,A -85,B 0,C 180,E1 -15195.411,E2 -15195.411} C_VEL
LIN {X 0,Y 319.722,Z 755.967,A -85,B 0,C 180,E1 -15197.3,E2 -15197.3} C_VEL
LIN {X 0,Y 318.896,Z 761.857,A -85,B 0,C 180,E1 -15199.201,E2 -15199.201} C_VEL
LIN {X 0,Y 318.347,Z 766.5,A -85,B 0,C 180,E1 -15201.108,E2 -15201.108} C_VEL
LIN {X 0,Y 318.112,Z 768.983,A -85,B 0,C 180,E1 -15202.381,E2 -15202.381} C_VEL
LIN {X 0,Y 317.977,Z 771.494,A -85,B 0,C 180,E1 -15204.047,E2 -15204.047} C_VEL
LIN {X 0,Y 317.991,Z 773.62,A -85,B 0,C 180,E1 -15206.196,E2 -15206.196} C_VEL
LIN {X 0,Y 318.008,Z 774.281,A -85,B 0,C 180,E1 -15207.465,E2 -15207.465} C_VEL
LIN {X 0,Y 318.185,Z 774.477,A -85,B 0,C 180,E1 -15208.732,E2 -15208.732} C_VEL
LIN {X 0,Y 318.269,Z 774.243,A -85,B 0,C 180,E1 -15209.998,E2 -15209.998} C_VEL
LIN {X 0,Y 318.247,Z 773.569,A -85,B 0,C 180,E1 -15211.263,E2 -15211.263} C_VEL
LIN {X 0,Y 318.117,Z 772.385,A -85,B 0,C 180,E1 -15212.53,E2 -15212.53} C_VEL
LIN {X 0,Y 318.108,Z 769.765,A -85,B 0,C 180,E1 -15214.433,E2 -15214.433} C_VEL
LIN {X 0,Y 318.12,Z 766.003,A -85,B 0,C 180,E1 -15216.34,E2 -15216.34} C_VEL
LIN {X 0,Y 318.225,Z 760.988,A -85,B 0,C 180,E1 -15218.251,E2 -15218.251} C_VEL
LIN {X 0,Y 318.538,Z 754.582,A -85,B 0,C 180,E1 -15220.164,E2 -15220.164} C_VEL
LIN {X 0,Y 319.113,Z 746.472,A -85,B 0,C 180,E1 -15222.075,E2 -15222.075} C_VEL
LIN {X 0,Y 319.75,Z 738.124,A -85,B 0,C 180,E1 -15223.665,E2 -15223.665} C_VEL
LIN {X 0,Y 320.337,Z 730.99,A -85,B 0,C 180,E1 -15224.805,E2 -15224.805} C_VEL
LIN {X 0,Y 321.447,Z 719.382,A -85,B 0,C 180,E1 -15226.331,E2 -15226.331} C_VEL
LIN {X 0,Y 322.336,Z 708.645,A -85,B 0,C 180,E1 -15227.443,E2 -15227.443} C_VEL
LIN {X 0,Y 323.323,Z 696.118,A -85,B 0,C 180,E1 -15228.452,E2 -15228.452} C_VEL
LIN {X 0,Y 324.962,Z 678.004,A -85,B 0,C 180,E1 -15229.83,E2 -15229.83} C_VEL
LIN {X 0,Y 325.889,Z 664.758,A -85,B 0,C 180,E1 -15230.553,E2 -15230.553} C_VEL
LIN {X 0,Y 326.448,Z 651.477,A -85,B 0,C 180,E1 -15231.011,E2 -15231.011} C_VEL
LIN {X 0,Y 327.276,Z 600.582,A -85,B 0,C 180,E1 -15232.133,E2 -15232.133} C_VEL
LIN {X 0,Y 322.356,Z 547.932,A -85,B 0,C 180,E1 -15233.649,E2 -15233.649} C_VEL
LIN {X 0,Y 322.141,Z 543.127,A -85,B 0,C 180,E1 -15233.943,E2 -15233.943} C_VEL
LIN {X 0,Y 324.3,Z 521.804,A -85,B 0,C 180,E1 -15238.119,E2 -15238.119} C_VEL
LIN {X 0,Y 325.329,Z 511.226,A -85,B 0,C 180,E1 -15240.218,E2 -15240.218} C_VEL
LIN {X 0,Y 322.469,Z 497.344,A -85,B 0,C 180,E1 -15243.288,E2 -15243.288} C_VEL
LIN {X 0,Y 319.642,Z 484.81,A -85,B 0,C 180,E1 -15246.244,E2 -15246.244} C_VEL
LIN {X 0,Y 319.521,Z 484.683,A -85,B 0,C 180,E1 -15249.66,E2 -15249.66} C_VEL
LIN {X 0,Y 319.512,Z 484.682,A -85,B 0,C 180,E1 -15253.458,E2 -15253.458} C_VEL
LIN {X 0,Y 319.544,Z 484.679,A -85,B 0,C 180,E1 -15257.014,E2 -15257.014} C_VEL
LIN {X 0,Y 319.535,Z 484.682,A -85,B 0,C 180,E1 -15260.369,E2 -15260.369} C_VEL
LIN {X 0,Y 319.569,Z 484.675,A -85,B 0,C 180,E1 -15264.455,E2 -15264.455} C_VEL
LIN {X 0,Y 319.522,Z 484.685,A -85,B 0,C 180,E1 -15268.137,E2 -15268.137} C_VEL
LIN {X 0,Y 319.604,Z 484.667,A -85,B 0,C 180,E1 -15271.587,E2 -15271.587} C_VEL
LIN {X 0,Y 319.593,Z 484.672,A -85,B 0,C 180,E1 -15275.303,E2 -15275.303} C_VEL
LIN {X 0,Y 319.585,Z 484.675,A -85,B 0,C 180,E1 -15278.046,E2 -15278.046} C_VEL
LIN {X 0,Y 319.677,Z 484.66,A -85,B 0,C 180,E1 -15280.961,E2 -15280.961} C_VEL
LIN {X 0,Y 319.718,Z 484.656,A -85,B 0,C 180,E1 -15285.275,E2 -15285.275} C_VEL
LIN {X 0,Y 319.745,Z 484.649,A -85,B 0,C 180,E1 -15289.872,E2 -15289.872} C_VEL
LIN {X 0,Y 319.919,Z 484.635,A -85,B 0,C 180,E1 -15292.425,E2 -15292.425} C_VEL
LIN {X 0,Y 319.732,Z 484.655,A -85,B 0,C 180,E1 -15294.955,E2 -15294.955} C_VEL
LIN {X 0,Y 319.976,Z 484.62,A -85,B 0,C 180,E1 -15297.482,E2 -15297.482} C_VEL
LIN {X 0,Y 320.136,Z 484.601,A -85,B 0,C 180,E1 -15300,E2 -15300} C_VEL
LIN {X 0,Y 319.977,Z 484.628,A -85,B 0,C 180,E1 -15302.517,E2 -15302.517} C_VEL
LIN {X 0,Y 319.914,Z 484.63,A -85,B 0,C 180,E1 -15306.715,E2 -15306.715} C_VEL
LIN {X 0,Y 319.744,Z 484.649,A -85,B 0,C 180,E1 -15310.127,E2 -15310.127} C_VEL
LIN {X 0,Y 319.717,Z 484.661,A -85,B 0,C 180,E1 -15314.724,E2 -15314.724} C_VEL
LIN {X 0,Y 319.675,Z 484.658,A -85,B 0,C 180,E1 -15319.038,E2 -15319.038} C_VEL
LIN {X 0,Y 319.556,Z 484.677,A -85,B 0,C 180,E1 -15323.32,E2 -15323.32} C_VEL
LIN {X 0,Y 319.621,Z 484.668,A -85,B 0,C 180,E1 -15326.089,E2 -15326.089} C_VEL
LIN {X 0,Y 319.576,Z 484.674,A -85,B 0,C 180,E1 -15328.934,E2 -15328.934} C_VEL
LIN {X 0,Y 319.519,Z 484.68,A -85,B 0,C 180,E1 -15331.863,E2 -15331.863} C_VEL
LIN {X 0,Y 319.567,Z 484.674,A -85,B 0,C 180,E1 -15335.544,E2 -15335.544} C_VEL
LIN {X 0,Y 319.546,Z 484.677,A -85,B 0,C 180,E1 -15339.67,E2 -15339.67} C_VEL
LIN {X 0,Y 319.552,Z 484.676,A -85,B 0,C 180,E1 -15343.47,E2 -15343.47} C_VEL
LIN {X 0,Y 319.592,Z 484.677,A -85,B 0,C 180,E1 -15347.026,E2 -15347.026} C_VEL
LIN {X 0,Y 319.577,Z 484.674,A -85,B 0,C 180,E1 -15350.379,E2 -15350.379} C_VEL
LIN {X 0,Y 319.552,Z 484.668,A -85,B 0,C 180,E1 -15353.575,E2 -15353.575} C_VEL
LIN {X 0,Y 319.568,Z 484.676,A -85,B 0,C 180,E1 -15356.688,E2 -15356.688} C_VEL
LIN {X 0,Y 319.583,Z 484.673,A -85,B 0,C 180,E1 -15359.618,E2 -15359.618} C_VEL
LIN {X 0,Y 319.6,Z 484.666,A -85,B 0,C 180,E1 -15362.5,E2 -15362.5} C_VEL
LIN {X 0,Y 319.598,Z 484.675,A -85,B 0,C 180,E1 -15365.306,E2 -15365.306} C_VEL
LIN {X 0,Y 319.59,Z 484.669,A -85,B 0,C 180,E1 -15368.05,E2 -15368.05} C_VEL
LIN {X 0,Y 319.683,Z 484.667,A -85,B 0,C 180,E1 -15370.964,E2 -15370.964} C_VEL
LIN {X 0,Y 319.726,Z 484.658,A -85,B 0,C 180,E1 -15375.278,E2 -15375.278} C_VEL
LIN {X 0,Y 319.754,Z 484.655,A -85,B 0,C 180,E1 -15379.875,E2 -15379.875} C_VEL
LIN {X 0,Y 319.843,Z 484.799,A -85,B 0,C 180,E1 -15380.867,E2 -15380.867} C_VEL
LIN {X 0,Y 320.123,Z 485.823,A -85,B 0,C 180,E1 -15381.087,E2 -15381.087} C_VEL
LIN {X 0,Y 327.259,Z 504.438,A -85,B 0,C 180,E1 -15381.973,E2 -15381.973} C_VEL
LIN {X 0,Y 328.363,Z 507.859,A -85,B 0,C 180,E1 -15382.118,E2 -15382.118} C_VEL
LIN {X 0,Y 327.561,Z 560.722,A -85,B 0,C 180,E1 -15383.28,E2 -15383.28} C_VEL
LIN {X 0,Y 327.476,Z 573.308,A -85,B 0,C 180,E1 -15383.669,E2 -15383.669} C_VEL
LIN {X 0,Y 327.197,Z 585.913,A -85,B 0,C 180,E1 -15384.301,E2 -15384.301} C_VEL
LIN {X 0,Y 326.609,Z 598.943,A -85,B 0,C 180,E1 -15385.219,E2 -15385.219} C_VEL
LIN {X 0,Y 325.883,Z 610.339,A -85,B 0,C 180,E1 -15386.293,E2 -15386.293} C_VEL
LIN {X 0,Y 324.936,Z 621.855,A -85,B 0,C 180,E1 -15387.678,E2 -15387.678} C_VEL
LIN {X 0,Y 324.059,Z 630.953,A -85,B 0,C 180,E1 -15389.036,E2 -15389.036} C_VEL
LIN {X 0,Y 323.034,Z 640.502,A -85,B 0,C 180,E1 -15390.797,E2 -15390.797} C_VEL
LIN {X 0,Y 322.074,Z 649.177,A -85,B 0,C 180,E1 -15392.816,E2 -15392.816} C_VEL
LIN {X 0,Y 321.418,Z 654.639,A -85,B 0,C 180,E1 -15394.391,E2 -15394.391} C_VEL
LIN {X 0,Y 320.837,Z 659.98,A -85,B 0,C 180,E1 -15396.29,E2 -15396.29} C_VEL
LIN {X 0,Y 320.384,Z 664.166,A -85,B 0,C 180,E1 -15398.2,E2 -15398.2} C_VEL
LIN {X 0,Y 320.034,Z 667.309,A -85,B 0,C 180,E1 -15400.12,E2 -15400.12} C_VEL
LIN {X 0,Y 319.925,Z 668.872,A -85,B 0,C 180,E1 -15401.405,E2 -15401.405} C_VEL
LIN {X 0,Y 319.861,Z 669.981,A -85,B 0,C 180,E1 -15402.695,E2 -15402.695} C_VEL
LIN {X 0,Y 320.014,Z 671.02,A -85,B 0,C 180,E1 -15405.282,E2 -15405.282} C_VEL
LIN {X 0,Y 320.197,Z 670.92,A -85,B 0,C 180,E1 -15406.581,E2 -15406.581} C_VEL
LIN {X 0,Y 320.437,Z 670.395,A -85,B 0,C 180,E1 -15407.884,E2 -15407.884} C_VEL
LIN {X 0,Y 320.943,Z 669.009,A -85,B 0,C 180,E1 -15409.677,E2 -15409.677} C_VEL
LIN {X 0,Y 321.742,Z 666.276,A -85,B 0,C 180,E1 -15411.8,E2 -15411.8} C_VEL
LIN {X 0,Y 322.723,Z 662.456,A -85,B 0,C 180,E1 -15413.846,E2 -15413.846} C_VEL
LIN {X 0,Y 323.846,Z 657.787,A -85,B 0,C 180,E1 -15415.726,E2 -15415.726} C_VEL
LIN {X 0,Y 325.41,Z 650.906,A -85,B 0,C 180,E1 -15417.868,E2 -15417.868} C_VEL
LIN {X 0,Y 326.852,Z 643.636,A -85,B 0,C 180,E1 -15419.642,E2 -15419.642} C_VEL
LIN {X 0,Y 328.539,Z 634.576,A -85,B 0,C 180,E1 -15421.411,E2 -15421.411} C_VEL
LIN {X 0,Y 329.968,Z 625.189,A -85,B 0,C 180,E1 -15422.899,E2 -15422.899} C_VEL
LIN {X 0,Y 331.439,Z 614.735,A -85,B 0,C 180,E1 -15424.211,E2 -15424.211} C_VEL
LIN {X 0,Y 332.667,Z 603.487,A -85,B 0,C 180,E1 -15425.335,E2 -15425.335} C_VEL
LIN {X 0,Y 333.515,Z 591.757,A -85,B 0,C 180,E1 -15426.254,E2 -15426.254} C_VEL
LIN {X 0,Y 334.183,Z 578.949,A -85,B 0,C 180,E1 -15426.973,E2 -15426.973} C_VEL
LIN {X 0,Y 334.368,Z 566.761,A -85,B 0,C 180,E1 -15427.434,E2 -15427.434} C_VEL
LIN {X 0,Y 335.026,Z 527.028,A -85,B 0,C 180,E1 -15428.351,E2 -15428.351} C_VEL
LIN {X 0,Y 335.244,Z 515.452,A -85,B 0,C 180,E1 -15428.612,E2 -15428.612} C_VEL
LIN {X 0,Y 326.524,Z 498.028,A -85,B 0,C 180,E1 -15429.938,E2 -15429.938} C_VEL
LIN {X 0,Y 323.943,Z 493.433,A -85,B 0,C 180,E1 -15430.333,E2 -15430.333} C_VEL
LIN {X 0,Y 321.667,Z 490.494,A -85,B 0,C 180,E1 -15430.677,E2 -15430.677} C_VEL
LIN {X 0,Y 317.981,Z 487.835,A -85,B 0,C 180,E1 -15431.277,E2 -15431.277} C_VEL
LIN {X 0,Y 314.601,Z 486.266,A -85,B 0,C 180,E1 -15432.03,E2 -15432.03} C_VEL
LIN {X 0,Y 312.879,Z 485.674,A -85,B 0,C 180,E1 -15432.704,E2 -15432.704} C_VEL
LIN {X 0,Y 312.462,Z 485.556,A -85,B 0,C 180,E1 -15433.195,E2 -15433.195} C_VEL
LIN {X 0,Y 312.498,Z 485.737,A -85,B 0,C 180,E1 -15435.148,E2 -15435.148} C_VEL
LIN {X 0,Y 315.964,Z 500.4,A -85,B 0,C 180,E1 -15438.402,E2 -15438.402} C_VEL
LIN {X 0,Y 318.128,Z 510.857,A -85,B 0,C 180,E1 -15440.646,E2 -15440.646} C_VEL
LIN {X 0,Y 318.196,Z 514.738,A -85,B 0,C 180,E1 -15441.413,E2 -15441.413} C_VEL
LIN {X 0,Y 317.545,Z 525.721,A -85,B 0,C 180,E1 -15443.494,E2 -15443.494} C_VEL
LIN {X 0,Y 321.083,Z 550.848,A -85,B 0,C 180,E1 -15444.469,E2 -15444.469} C_VEL
LIN {X 0,Y 318.339,Z 637.624,A -85,B 0,C 180,E1 -15446.994,E2 -15446.994} C_VEL
LIN {X 0,Y 317.653,Z 651.061,A -85,B 0,C 180,E1 -15447.643,E2 -15447.643} C_VEL
LIN {X 0,Y 316.826,Z 664.671,A -85,B 0,C 180,E1 -15448.582,E2 -15448.582} C_VEL
LIN {X 0,Y 315.99,Z 676.86,A -85,B 0,C 180,E1 -15449.711,E2 -15449.711} C_VEL
LIN {X 0,Y 315.047,Z 687.738,A -85,B 0,C 180,E1 -15450.975,E2 -15450.975} C_VEL
LIN {X 0,Y 314.053,Z 698.365,A -85,B 0,C 180,E1 -15452.513,E2 -15452.513} C_VEL
LIN {X 0,Y 313.21,Z 707.711,A -85,B 0,C 180,E1 -15454.183,E2 -15454.183} C_VEL
LIN {X 0,Y 312.42,Z 716.462,A -85,B 0,C 180,E1 -15456.115,E2 -15456.115} C_VEL
LIN {X 0,Y 311.75,Z 723.825,A -85,B 0,C 180,E1 -15458.163,E2 -15458.163} C_VEL
LIN {X 0,Y 311.299,Z 729.62,A -85,B 0,C 180,E1 -15460.206,E2 -15460.206} C_VEL
LIN {X 0,Y 310.999,Z 734.018,A -85,B 0,C 180,E1 -15462.25,E2 -15462.25} C_VEL
LIN {X 0,Y 310.772,Z 737.156,A -85,B 0,C 180,E1 -15464.254,E2 -15464.254} C_VEL
LIN {X 0,Y 310.816,Z 739.373,A -85,B 0,C 180,E1 -15466.488,E2 -15466.488} C_VEL
LIN {X 0,Y 310.86,Z 740.225,A -85,B 0,C 180,E1 -15468.26,E2 -15468.26} C_VEL
LIN {X 0,Y 310.962,Z 740.342,A -85,B 0,C 180,E1 -15469.584,E2 -15469.584} C_VEL
LIN {X 0,Y 311.187,Z 740.031,A -85,B 0,C 180,E1 -15470.904,E2 -15470.904} C_VEL
LIN {X 0,Y 311.651,Z 738.712,A -85,B 0,C 180,E1 -15472.869,E2 -15472.869} C_VEL
LIN {X 0,Y 312.471,Z 735.367,A -85,B 0,C 180,E1 -15475.485,E2 -15475.485} C_VEL
LIN {X 0,Y 313.256,Z 731.656,A -85,B 0,C 180,E1 -15477.429,E2 -15477.429} C_VEL
LIN {X 0,Y 314.396,Z 726.801,A -85,B 0,C 180,E1 -15479.36,E2 -15479.36} C_VEL
LIN {X 0,Y 315.782,Z 720.626,A -85,B 0,C 180,E1 -15481.276,E2 -15481.276} C_VEL
LIN {X 0,Y 317.584,Z 712.384,A -85,B 0,C 180,E1 -15483.284,E2 -15483.284} C_VEL
LIN {X 0,Y 319.408,Z 703.27,A -85,B 0,C 180,E1 -15485.05,E2 -15485.05} C_VEL
LIN {X 0,Y 321.414,Z 692.262,A -85,B 0,C 180,E1 -15486.75,E2 -15486.75} C_VEL
LIN {X 0,Y 323.21,Z 680.987,A -85,B 0,C 180,E1 -15488.126,E2 -15488.126} C_VEL
LIN {X 0,Y 324.704,Z 670.049,A -85,B 0,C 180,E1 -15489.186,E2 -15489.186} C_VEL
LIN {X 0,Y 326.077,Z 658.104,A -85,B 0,C 180,E1 -15490.086,E2 -15490.086} C_VEL
LIN {X 0,Y 327.199,Z 644.553,A -85,B 0,C 180,E1 -15490.833,E2 -15490.833} C_VEL
LIN {X 0,Y 328.229,Z 626.943,A -85,B 0,C 180,E1 -15491.463,E2 -15491.463} C_VEL
LIN {X 0,Y 332.76,Z 556.791,A -85,B 0,C 180,E1 -15493.697,E2 -15493.697} C_VEL
LIN {X 0,Y 330.727,Z 545.376,A -85,B 0,C 180,E1 -15494.498,E2 -15494.498} C_VEL
LIN {X 0,Y 327.338,Z 530.878,A -85,B 0,C 180,E1 -15495.734,E2 -15495.734} C_VEL
LIN {X 0,Y 326.952,Z 526.926,A -85,B 0,C 180,E1 -15496.712,E2 -15496.712} C_VEL
LIN {X 0,Y 325.438,Z 518.994,A -85,B 0,C 180,E1 -15498.901,E2 -15498.901} C_VEL
LIN {X 0,Y 323.303,Z 511.152,A -85,B 0,C 180,E1 -15501.345,E2 -15501.345} C_VEL
LIN {X 0,Y 320.218,Z 502.193,A -85,B 0,C 180,E1 -15504.646,E2 -15504.646} C_VEL
LIN {X 0,Y 317.83,Z 496.683,A -85,B 0,C 180,E1 -15507.042,E2 -15507.042} C_VEL
LIN {X 0,Y 316.477,Z 493.583,A -85,B 0,C 180,E1 -15508.598,E2 -15508.598} C_VEL
LIN {X 0,Y 314.561,Z 489.745,A -85,B 0,C 180,E1 -15510.923,E2 -15510.923} C_VEL
LIN {X 0,Y 312.659,Z 486.262,A -85,B 0,C 180,E1 -15513.724,E2 -15513.724} C_VEL
LIN {X 0,Y 312.535,Z 485.644,A -85,B 0,C 180,E1 -15514.597,E2 -15514.597} C_VEL
LIN {X 0,Y 312.502,Z 485.555,A -85,B 0,C 180,E1 -15518.079,E2 -15518.079} C_VEL
LIN {X 0,Y 312.499,Z 485.556,A -85,B 0,C 180,E1 -15520.708,E2 -15520.708} C_VEL
LIN {X 0,Y 312.46,Z 485.56,A -85,B 0,C 180,E1 -15524.209,E2 -15524.209} C_VEL
LIN {X 0,Y 312.568,Z 485.973,A -85,B 0,C 180,E1 -15526.528,E2 -15526.528} C_VEL
LIN {X 0,Y 313.87,Z 488.959,A -85,B 0,C 180,E1 -15528.601,E2 -15528.601} C_VEL
LIN {X 0,Y 314.755,Z 490.007,A -85,B 0,C 180,E1 -15529.392,E2 -15529.392} C_VEL
LIN {X 0,Y 315.993,Z 496.021,A -85,B 0,C 180,E1 -15531.481,E2 -15531.481} C_VEL
LIN {X 0,Y 318.039,Z 503.953,A -85,B 0,C 180,E1 -15533.762,E2 -15533.762} C_VEL
LIN {X 0,Y 321.089,Z 514.697,A -85,B 0,C 180,E1 -15536.279,E2 -15536.279} C_VEL
LIN {X 0,Y 323.245,Z 522.073,A -85,B 0,C 180,E1 -15537.735,E2 -15537.735} C_VEL
LIN {X 0,Y 323.862,Z 526.723,A -85,B 0,C 180,E1 -15538.411,E2 -15538.411} C_VEL
LIN {X 0,Y 324.651,Z 543.361,A -85,B 0,C 180,E1 -15540.326,E2 -15540.326} C_VEL
LIN {X 0,Y 325.139,Z 550.731,A -85,B 0,C 180,E1 -15541.055,E2 -15541.055} C_VEL
LIN {X 0,Y 327.823,Z 570.237,A -85,B 0,C 180,E1 -15542.362,E2 -15542.362} C_VEL
LIN {X 0,Y 329.239,Z 587.732,A -85,B 0,C 180,E1 -15543.321,E2 -15543.321} C_VEL
LIN {X 0,Y 329.694,Z 605.627,A -85,B 0,C 180,E1 -15544.13,E2 -15544.13} C_VEL
LIN {X 0,Y 325.57,Z 672.289,A -85,B 0,C 180,E1 -15546.291,E2 -15546.291} C_VEL
LIN {X 0,Y 324.51,Z 684.225,A -85,B 0,C 180,E1 -15546.885,E2 -15546.885} C_VEL
LIN {X 0,Y 322.752,Z 697.429,A -85,B 0,C 180,E1 -15547.767,E2 -15547.767} C_VEL
LIN {X 0,Y 320.839,Z 710.715,A -85,B 0,C 180,E1 -15548.978,E2 -15548.978} C_VEL
LIN {X 0,Y 318.641,Z 723.616,A -85,B 0,C 180,E1 -15550.511,E2 -15550.511} C_VEL
LIN {X 0,Y 316.974,Z 733.06,A -85,B 0,C 180,E1 -15551.914,E2 -15551.914} C_VEL
LIN {X 0,Y 315.073,Z 743.012,A -85,B 0,C 180,E1 -15553.754,E2 -15553.754} C_VEL
LIN {X 0,Y 313.675,Z 751.523,A -85,B 0,C 180,E1 -15555.73,E2 -15555.73} C_VEL
LIN {X 0,Y 312.441,Z 758.186,A -85,B 0,C 180,E1 -15557.659,E2 -15557.659} C_VEL
LIN {X 0,Y 311.671,Z 763.532,A -85,B 0,C 180,E1 -15559.605,E2 -15559.605} C_VEL
LIN {X 0,Y 311.15,Z 767.687,A -85,B 0,C 180,E1 -15561.555,E2 -15561.555} C_VEL
LIN {X 0,Y 310.874,Z 771.523,A -85,B 0,C 180,E1 -15564.112,E2 -15564.112} C_VEL
LIN {X 0,Y 310.913,Z 773.301,A -85,B 0,C 180,E1 -15566.109,E2 -15566.109} C_VEL
LIN {X 0,Y 310.918,Z 773.879,A -85,B 0,C 180,E1 -15567.407,E2 -15567.407} C_VEL
LIN {X 0,Y 311.088,Z 774.034,A -85,B 0,C 180,E1 -15568.703,E2 -15568.703} C_VEL
LIN {X 0,Y 311.207,Z 773.759,A -85,B 0,C 180,E1 -15569.998,E2 -15569.998} C_VEL
LIN {X 0,Y 311.184,Z 772.999,A -85,B 0,C 180,E1 -15571.292,E2 -15571.292} C_VEL
LIN {X 0,Y 311.029,Z 771.757,A -85,B 0,C 180,E1 -15572.588,E2 -15572.588} C_VEL
LIN {X 0,Y 311.042,Z 769.036,A -85,B 0,C 180,E1 -15574.534,E2 -15574.534} C_VEL
LIN {X 0,Y 311.029,Z 765.159,A -85,B 0,C 180,E1 -15576.485,E2 -15576.485} C_VEL
LIN {X 0,Y 311.175,Z 760.029,A -85,B 0,C 180,E1 -15578.44,E2 -15578.44} C_VEL
LIN {X 0,Y 311.507,Z 753.465,A -85,B 0,C 180,E1 -15580.396,E2 -15580.396} C_VEL
LIN {X 0,Y 312.128,Z 745.173,A -85,B 0,C 180,E1 -15582.349,E2 -15582.349} C_VEL
LIN {X 0,Y 312.834,Z 736.662,A -85,B 0,C 180,E1 -15583.973,E2 -15583.973} C_VEL
LIN {X 0,Y 313.714,Z 726.144,A -85,B 0,C 180,E1 -15585.592,E2 -15585.592} C_VEL
LIN {X 0,Y 314.646,Z 715.773,A -85,B 0,C 180,E1 -15586.878,E2 -15586.878} C_VEL
LIN {X 0,Y 315.666,Z 704.525,A -85,B 0,C 180,E1 -15587.991,E2 -15587.991} C_VEL
LIN {X 0,Y 316.956,Z 688.962,A -85,B 0,C 180,E1 -15589.256,E2 -15589.256} C_VEL
LIN {X 0,Y 318.123,Z 676.803,A -85,B 0,C 180,E1 -15590.191,E2 -15590.191} C_VEL
LIN {X 0,Y 319.029,Z 664.335,A -85,B 0,C 180,E1 -15590.889,E2 -15590.889} C_VEL
LIN {X 0,Y 319.619,Z 651.437,A -85,B 0,C 180,E1 -15591.355,E2 -15591.355} C_VEL
LIN {X 0,Y 320.431,Z 600.427,A -85,B 0,C 180,E1 -15592.51,E2 -15592.51} C_VEL
LIN {X 0,Y 315.42,Z 546.302,A -85,B 0,C 180,E1 -15594.105,E2 -15594.105} C_VEL
LIN {X 0,Y 315.256,Z 542.116,A -85,B 0,C 180,E1 -15594.388,E2 -15594.388} C_VEL
LIN {X 0,Y 317.602,Z 520.31,A -85,B 0,C 180,E1 -15598.767,E2 -15598.767} C_VEL
LIN {X 0,Y 318.388,Z 513.516,A -85,B 0,C 180,E1 -15600.141,E2 -15600.141} C_VEL
LIN {X 0,Y 317.152,Z 506.258,A -85,B 0,C 180,E1 -15601.752,E2 -15601.752} C_VEL
LIN {X 0,Y 313.754,Z 490.624,A -85,B 0,C 180,E1 -15605.393,E2 -15605.393} C_VEL
LIN {X 0,Y 312.561,Z 485.674,A -85,B 0,C 180,E1 -15606.641,E2 -15606.641} C_VEL
LIN {X 0,Y 312.433,Z 485.565,A -85,B 0,C 180,E1 -15610.715,E2 -15610.715} C_VEL
LIN {X 0,Y 312.443,Z 485.567,A -85,B 0,C 180,E1 -15614.208,E2 -15614.208} C_VEL
LIN {X 0,Y 312.474,Z 485.562,A -85,B 0,C 180,E1 -15617.917,E2 -15617.917} C_VEL
LIN {X 0,Y 312.467,Z 485.56,A -85,B 0,C 180,E1 -15620.966,E2 -15620.966} C_VEL
LIN {X 0,Y 312.521,Z 485.555,A -85,B 0,C 180,E1 -15624.218,E2 -15624.218} C_VEL
LIN {X 0,Y 312.494,Z 485.556,A -85,B 0,C 180,E1 -15627.332,E2 -15627.332} C_VEL
LIN {X 0,Y 312.54,Z 485.546,A -85,B 0,C 180,E1 -15631.275,E2 -15631.275} C_VEL
LIN {X 0,Y 312.573,Z 485.549,A -85,B 0,C 180,E1 -15634.709,E2 -15634.709} C_VEL
LIN {X 0,Y 312.575,Z 485.546,A -85,B 0,C 180,E1 -15637.528,E2 -15637.528} C_VEL
LIN {X 0,Y 312.626,Z 485.537,A -85,B 0,C 180,E1 -15641.655,E2 -15641.655} C_VEL
LIN {X 0,Y 312.681,Z 485.533,A -85,B 0,C 180,E1 -15645.685,E2 -15645.685} C_VEL
LIN {X 0,Y 312.689,Z 485.526,A -85,B 0,C 180,E1 -15649.641,E2 -15649.641} C_VEL
LIN {X 0,Y 312.858,Z 485.513,A -85,B 0,C 180,E1 -15652.253,E2 -15652.253} C_VEL
LIN {X 0,Y 312.702,Z 485.532,A -85,B 0,C 180,E1 -15654.842,E2 -15654.842} C_VEL
LIN {X 0,Y 312.977,Z 485.493,A -85,B 0,C 180,E1 -15658.713,E2 -15658.713} C_VEL
LIN {X 0,Y 312.979,Z 485.494,A -85,B 0,C 180,E1 -15661.286,E2 -15661.286} C_VEL
LIN {X 0,Y 312.703,Z 485.53,A -85,B 0,C 180,E1 -15665.157,E2 -15665.157} C_VEL
LIN {X 0,Y 312.857,Z 485.506,A -85,B 0,C 180,E1 -15667.746,E2 -15667.746} C_VEL
LIN {X 0,Y 312.656,Z 485.534,A -85,B 0,C 180,E1 -15671.671,E2 -15671.671} C_VEL
LIN {X 0,Y 312.686,Z 485.535,A -85,B 0,C 180,E1 -15674.888,E2 -15674.888} C_VEL
LIN {X 0,Y 312.617,Z 485.535,A -85,B 0,C 180,E1 -15679.237,E2 -15679.237} C_VEL
LIN {X 0,Y 312.532,Z 485.556,A -85,B 0,C 180,E1 -15682.79,E2 -15682.79} C_VEL
LIN {X 0,Y 312.569,Z 485.549,A -85,B 0,C 180,E1 -15686.723,E2 -15686.723} C_VEL
LIN {X 0,Y 312.532,Z 485.547,A -85,B 0,C 180,E1 -15689.651,E2 -15689.651} C_VEL
LIN {X 0,Y 312.506,Z 485.555,A -85,B 0,C 180,E1 -15693.69,E2 -15693.69} C_VEL
LIN {X 0,Y 312.508,Z 485.551,A -85,B 0,C 180,E1 -15697.387,E2 -15697.387} C_VEL
LIN {X 0,Y 312.478,Z 485.562,A -85,B 0,C 180,E1 -15700.71,E2 -15700.71} C_VEL
LIN {X 0,Y 312.507,Z 485.553,A -85,B 0,C 180,E1 -15704.199,E2 -15704.199} C_VEL
LIN {X 0,Y 312.538,Z 485.551,A -85,B 0,C 180,E1 -15707.907,E2 -15707.907} C_VEL
LIN {X 0,Y 312.551,Z 485.542,A -85,B 0,C 180,E1 -15711.906,E2 -15711.906} C_VEL
LIN {X 0,Y 312.497,Z 485.553,A -85,B 0,C 180,E1 -15715.792,E2 -15715.792} C_VEL
LIN {X 0,Y 312.515,Z 485.559,A -85,B 0,C 180,E1 -15718.856,E2 -15718.856} C_VEL
LIN {X 0,Y 312.566,Z 485.54,A -85,B 0,C 180,E1 -15721.827,E2 -15721.827} C_VEL
LIN {X 0,Y 312.578,Z 485.547,A -85,B 0,C 180,E1 -15724.713,E2 -15724.713} C_VEL
LIN {X 0,Y 312.581,Z 485.543,A -85,B 0,C 180,E1 -15727.531,E2 -15727.531} C_VEL
LIN {X 0,Y 312.632,Z 485.54,A -85,B 0,C 180,E1 -15731.658,E2 -15731.658} C_VEL
LIN {X 0,Y 312.689,Z 485.532,A -85,B 0,C 180,E1 -15735.688,E2 -15735.688} C_VEL
LIN {X 0,Y 312.753,Z 485.583,A -85,B 0,C 180,E1 -15740.324,E2 -15740.324} C_VEL
LIN {X 0,Y 312.915,Z 486.351,A -85,B 0,C 180,E1 -15740.598,E2 -15740.598} C_VEL
LIN {X 0,Y 318.754,Z 500.932,A -85,B 0,C 180,E1 -15741.366,E2 -15741.366} C_VEL
LIN {X 0,Y 321.573,Z 508.923,A -85,B 0,C 180,E1 -15741.731,E2 -15741.731} C_VEL
LIN {X 0,Y 320.815,Z 561.194,A -85,B 0,C 180,E1 -15742.907,E2 -15742.907} C_VEL
LIN {X 0,Y 320.687,Z 574.788,A -85,B 0,C 180,E1 -15743.337,E2 -15743.337} C_VEL
LIN {X 0,Y 320.355,Z 587.89,A -85,B 0,C 180,E1 -15744.021,E2 -15744.021} C_VEL
LIN {X 0,Y 319.789,Z 600.628,A -85,B 0,C 180,E1 -15744.959,E2 -15744.959} C_VEL
LIN {X 0,Y 319.007,Z 611.863,A -85,B 0,C 180,E1 -15746.054,E2 -15746.054} C_VEL
LIN {X 0,Y 318.034,Z 623.284,A -85,B 0,C 180,E1 -15747.469,E2 -15747.469} C_VEL
LIN {X 0,Y 317.061,Z 633.131,A -85,B 0,C 180,E1 -15748.997,E2 -15748.997} C_VEL
LIN {X 0,Y 316.123,Z 641.393,A -85,B 0,C 180,E1 -15750.575,E2 -15750.575} C_VEL
LIN {X 0,Y 315.148,Z 649.783,A -85,B 0,C 180,E1 -15752.558,E2 -15752.558} C_VEL
LIN {X 0,Y 314.341,Z 656.322,A -85,B 0,C 180,E1 -15754.49,E2 -15754.49} C_VEL
LIN {X 0,Y 313.766,Z 661.524,A -85,B 0,C 180,E1 -15756.432,E2 -15756.432} C_VEL
LIN {X 0,Y 313.319,Z 665.584,A -85,B 0,C 180,E1 -15758.386,E2 -15758.386} C_VEL
LIN {X 0,Y 312.969,Z 668.615,A -85,B 0,C 180,E1 -15760.351,E2 -15760.351} C_VEL
LIN {X 0,Y 312.868,Z 670.07,A -85,B 0,C 180,E1 -15761.666,E2 -15761.666} C_VEL
LIN {X 0,Y 312.899,Z 671.778,A -85,B 0,C 180,E1 -15764.306,E2 -15764.306} C_VEL
LIN {X 0,Y 313.037,Z 672.027,A -85,B 0,C 180,E1 -15765.631,E2 -15765.631} C_VEL
LIN {X 0,Y 313.229,Z 671.841,A -85,B 0,C 180,E1 -15766.961,E2 -15766.961} C_VEL
LIN {X 0,Y 313.511,Z 671.26,A -85,B 0,C 180,E1 -15768.293,E2 -15768.293} C_VEL
LIN {X 0,Y 314.009,Z 669.95,A -85,B 0,C 180,E1 -15769.946,E2 -15769.946} C_VEL
LIN {X 0,Y 314.963,Z 666.909,A -85,B 0,C 180,E1 -15772.294,E2 -15772.294} C_VEL
LIN {X 0,Y 315.93,Z 663.335,A -85,B 0,C 180,E1 -15774.209,E2 -15774.209} C_VEL
LIN {X 0,Y 317.25,Z 658.16,A -85,B 0,C 180,E1 -15776.301,E2 -15776.301} C_VEL
LIN {X 0,Y 318.789,Z 651.583,A -85,B 0,C 180,E1 -15778.347,E2 -15778.347} C_VEL
LIN {X 0,Y 320.436,Z 643.601,A -85,B 0,C 180,E1 -15780.297,E2 -15780.297} C_VEL
LIN {X 0,Y 322.101,Z 635.15,A -85,B 0,C 180,E1 -15781.948,E2 -15781.948} C_VEL
LIN {X 0,Y 323.588,Z 625.773,A -85,B 0,C 180,E1 -15783.446,E2 -15783.446} C_VEL
LIN {X 0,Y 325.099,Z 615.344,A -85,B 0,C 180,E1 -15784.767,E2 -15784.767} C_VEL
LIN {X 0,Y 326.41,Z 603.816,A -85,B 0,C 180,E1 -15785.927,E2 -15785.927} C_VEL
LIN {X 0,Y 327.324,Z 591.861,A -85,B 0,C 180,E1 -15786.861,E2 -15786.861} C_VEL
LIN {X 0,Y 327.947,Z 578.802,A -85,B 0,C 180,E1 -15787.588,E2 -15787.588} C_VEL
LIN {X 0,Y 328.142,Z 566.074,A -85,B 0,C 180,E1 -15788.053,E2 -15788.053} C_VEL
LIN {X 0,Y 328.9,Z 526.059,A -85,B 0,C 180,E1 -15788.981,E2 -15788.981} C_VEL
LIN {X 0,Y 328.995,Z 517.436,A -85,B 0,C 180,E1 -15789.188,E2 -15789.188} C_VEL
LIN {X 0,Y 320.953,Z 501.477,A -85,B 0,C 180,E1 -15790.455,E2 -15790.455} C_VEL
LIN {X 0,Y 313.633,Z 488.547,A -85,B 0,C 180,E1 -15791.644,E2 -15791.644} C_VEL
LIN {X 0,Y 312.617,Z 486.128,A -85,B 0,C 180,E1 -15791.93,E2 -15791.93} C_VEL
LIN {X 0,Y 312.517,Z 485.629,A -85,B 0,C 180,E1 -15792.202,E2 -15792.202} C_VEL
LIN {X 0,Y 312.462,Z 485.556,A -85,B 0,C 180,E1 -15793.195,E2 -15793.195} C_VEL
LIN {X 0,Y 312.215,Z 486.011,A -85,B 0,C 180,E1 -15793.901,E2 -15793.901} C_VEL
LIN {X 0,Y 311.287,Z 488.001,A -85,B 0,C 180,E1 -15794.902,E2 -15794.902} C_VEL
LIN {X 0,Y 310.119,Z 491.031,A -85,B 0,C 180,E1 -15795.819,E2 -15795.819} C_VEL
LIN {X 0,Y 308.858,Z 496.122,A -85,B 0,C 180,E1 -15796.987,E2 -15796.987} C_VEL
LIN {X 0,Y 308.765,Z 500.161,A -85,B 0,C 180,E1 -15797.841,E2 -15797.841} C_VEL
LIN {X 0,Y 308.996,Z 501.481,A -85,B 0,C 180,E1 -15798.127,E2 -15798.127} C_VEL
LIN {X 0,Y 311.32,Z 512.925,A -85,B 0,C 180,E1 -15800.587,E2 -15800.587} C_VEL
LIN {X 0,Y 310.946,Z 522.039,A -85,B 0,C 180,E1 -15802.393,E2 -15802.393} C_VEL
LIN {X 0,Y 310.668,Z 526.206,A -85,B 0,C 180,E1 -15803.145,E2 -15803.145} C_VEL
LIN {X 0,Y 314.187,Z 551.98,A -85,B 0,C 180,E1 -15804.162,E2 -15804.162} C_VEL
LIN {X 0,Y 311.385,Z 637.838,A -85,B 0,C 180,E1 -15806.731,E2 -15806.731} C_VEL
LIN {X 0,Y 310.807,Z 650.179,A -85,B 0,C 180,E1 -15807.326,E2 -15807.326} C_VEL
LIN {X 0,Y 309.937,Z 663.987,A -85,B 0,C 180,E1 -15808.279,E2 -15808.279} C_VEL
LIN {X 0,Y 309.075,Z 676.328,A -85,B 0,C 180,E1 -15809.419,E2 -15809.419} C_VEL
LIN {X 0,Y 308.023,Z 688.147,A -85,B 0,C 180,E1 -15810.811,E2 -15810.811} C_VEL
LIN {X 0,Y 307.003,Z 698.778,A -85,B 0,C 180,E1 -15812.383,E2 -15812.383} C_VEL
